REGION Network 33: Interface Signals 05 -Example: Model Flex-Pro-Line - IN/OUT- / Interface Signals 28
   // Aufruf des Schnittstellen Signal Bausteins Ba-Bereich 4 / Call the interface signals bool blocks of opmode 4
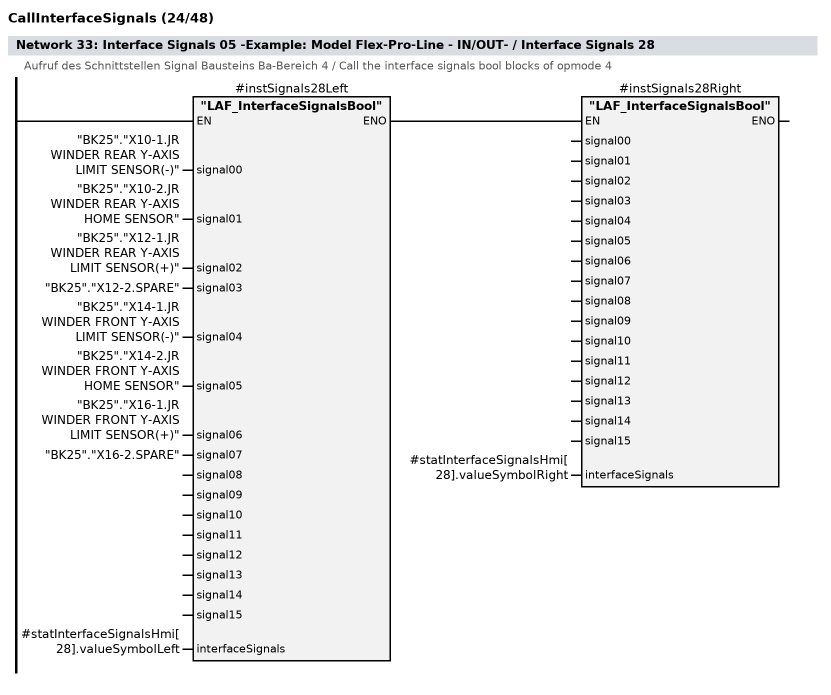
   RUNG wire#powerrail
      #instSignals28Left(signal00 := "BK25"."X10-1.JR WINDER REAR Y-AXIS LIMIT SENSOR(-)", signal01 := "BK25"."X10-2.JR WINDER REAR Y-AXIS HOME SENSOR", signal02 := "BK25"."X12-1.JR WINDER REAR Y-AXIS LIMIT SENSOR(+)", signal03 := "BK25"."X12-2.SPARE", signal04 := "BK25"."X14-1.JR WINDER FRONT Y-AXIS LIMIT SENSOR(-)", signal05 := "BK25"."X14-2.JR WINDER FRONT Y-AXIS HOME SENSOR", signal06 := "BK25"."X16-1.JR WINDER FRONT Y-AXIS LIMIT SENSOR(+)", signal07 := "BK25"."X16-2.SPARE", signal08 :=, signal09 :=, signal10 :=, signal11 :=, signal12 :=, signal13 :=, signal14 :=, signal15 :=, interfaceSignals := #statInterfaceSignalsHmi[28].valueSymbolLeft)
      #instSignals28Right(signal00 :=, signal01 :=, signal02 :=, signal03 :=, signal04 :=, signal05 :=, signal06 :=, signal07 :=, signal08 :=, signal09 :=, signal10 :=, signal11 :=, signal12 :=, signal13 :=, signal14 :=, signal15 :=, interfaceSignals := #statInterfaceSignalsHmi[28].valueSymbolRight)
   END_RUNG
   // the same network as SCL:
   #instSignals28Left(signal00 := "BK25"."X10-1.JR WINDER REAR Y-AXIS LIMIT SENSOR(-)",   // "LAF_InterfaceSignalsBool"
                      signal01 := "BK25"."X10-2.JR WINDER REAR Y-AXIS HOME SENSOR",
                      signal02 := "BK25"."X12-1.JR WINDER REAR Y-AXIS LIMIT SENSOR(+)",
                      signal03 := "BK25"."X12-2.SPARE",
                      signal04 := "BK25"."X14-1.JR WINDER FRONT Y-AXIS LIMIT SENSOR(-)",
                      signal05 := "BK25"."X14-2.JR WINDER FRONT Y-AXIS HOME SENSOR",
                      signal06 := "BK25"."X16-1.JR WINDER FRONT Y-AXIS LIMIT SENSOR(+)",
                      signal07 := "BK25"."X16-2.SPARE",
                      interfaceSignals := #statInterfaceSignalsHmi[28].valueSymbolLeft,
                      ENO => #_w1);
   IF #_w1 THEN
       #instSignals28Right(interfaceSignals := #statInterfaceSignalsHmi[28].valueSymbolRight);   // "LAF_InterfaceSignalsBool"
   END_IF;
END_REGION

REGION Network 34: Interface Signals 05 -Example: Model Flex-Pro-Line - IN/OUT- / Interface Signals 29
   // Aufruf des Schnittstellen Signal Bausteins Ba-Bereich 4 / Call the interface signals bool blocks of opmode 4
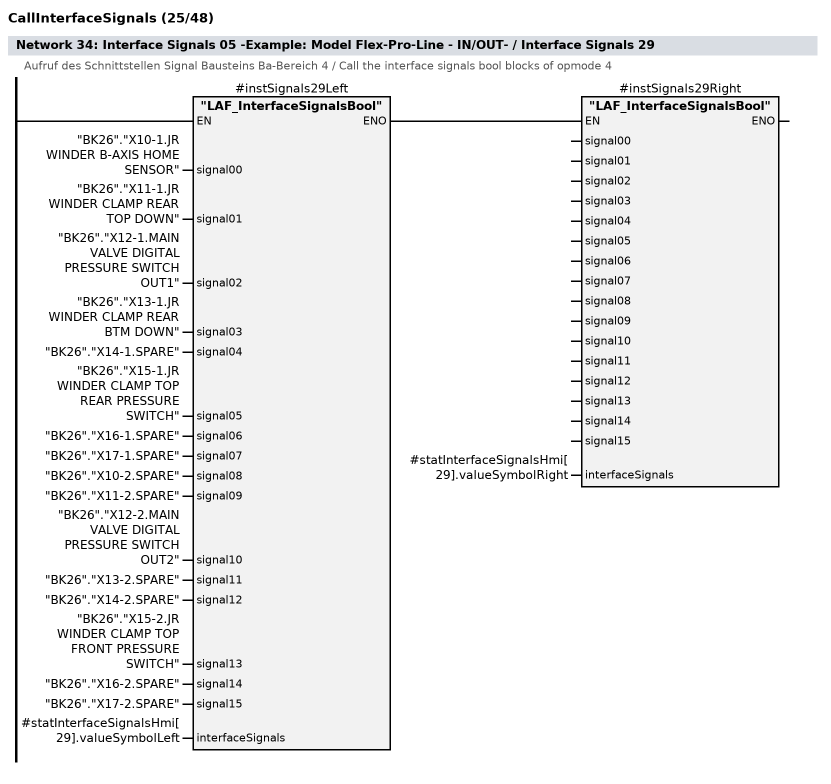
   RUNG wire#powerrail
      #instSignals29Left(signal00 := "BK26"."X10-1.JR WINDER B-AXIS HOME SENSOR", signal01 := "BK26"."X11-1.JR WINDER CLAMP REAR TOP DOWN", signal02 := "BK26"."X12-1.MAIN VALVE DIGITAL PRESSURE SWITCH OUT1", signal03 := "BK26"."X13-1.JR WINDER CLAMP REAR BTM DOWN", signal04 := "BK26"."X14-1.SPARE", signal05 := "BK26"."X15-1.JR WINDER CLAMP TOP REAR PRESSURE SWITCH", signal06 := "BK26"."X16-1.SPARE", signal07 := "BK26"."X17-1.SPARE", signal08 := "BK26"."X10-2.SPARE", signal09 := "BK26"."X11-2.SPARE", signal10 := "BK26"."X12-2.MAIN VALVE DIGITAL PRESSURE SWITCH OUT2", signal11 := "BK26"."X13-2.SPARE", signal12 := "BK26"."X14-2.SPARE", signal13 := "BK26"."X15-2.JR WINDER CLAMP TOP FRONT PRESSURE SWITCH", signal14 := "BK26"."X16-2.SPARE", signal15 := "BK26"."X17-2.SPARE", interfaceSignals := #statInterfaceSignalsHmi[29].valueSymbolLeft)
      #instSignals29Right(signal00 :=, signal01 :=, signal02 :=, signal03 :=, signal04 :=, signal05 :=, signal06 :=, signal07 :=, signal08 :=, signal09 :=, signal10 :=, signal11 :=, signal12 :=, signal13 :=, signal14 :=, signal15 :=, interfaceSignals := #statInterfaceSignalsHmi[29].valueSymbolRight)
   END_RUNG
   // the same network as SCL:
   #instSignals29Left(signal00 := "BK26"."X10-1.JR WINDER B-AXIS HOME SENSOR",   // "LAF_InterfaceSignalsBool"
                      signal01 := "BK26"."X11-1.JR WINDER CLAMP REAR TOP DOWN",
                      signal02 := "BK26"."X12-1.MAIN VALVE DIGITAL PRESSURE SWITCH OUT1",
                      signal03 := "BK26"."X13-1.JR WINDER CLAMP REAR BTM DOWN",
                      signal04 := "BK26"."X14-1.SPARE",
                      signal05 := "BK26"."X15-1.JR WINDER CLAMP TOP REAR PRESSURE SWITCH",
                      signal06 := "BK26"."X16-1.SPARE",
                      signal07 := "BK26"."X17-1.SPARE",
                      signal08 := "BK26"."X10-2.SPARE",
                      signal09 := "BK26"."X11-2.SPARE",
                      signal10 := "BK26"."X12-2.MAIN VALVE DIGITAL PRESSURE SWITCH OUT2",
                      signal11 := "BK26"."X13-2.SPARE",
                      signal12 := "BK26"."X14-2.SPARE",
                      signal13 := "BK26"."X15-2.JR WINDER CLAMP TOP FRONT PRESSURE SWITCH",
                      signal14 := "BK26"."X16-2.SPARE",
                      signal15 := "BK26"."X17-2.SPARE",
                      interfaceSignals := #statInterfaceSignalsHmi[29].valueSymbolLeft,
                      ENO => #_w1);
   IF #_w1 THEN
       #instSignals29Right(interfaceSignals := #statInterfaceSignalsHmi[29].valueSymbolRight);   // "LAF_InterfaceSignalsBool"
   END_IF;
END_REGION

REGION Network 35: Interface Signals 05 -Example: Model Flex-Pro-Line - IN/OUT- / Interface Signals 30
   // Aufruf des Schnittstellen Signal Bausteins Ba-Bereich 4 / Call the interface signals bool blocks of opmode 4
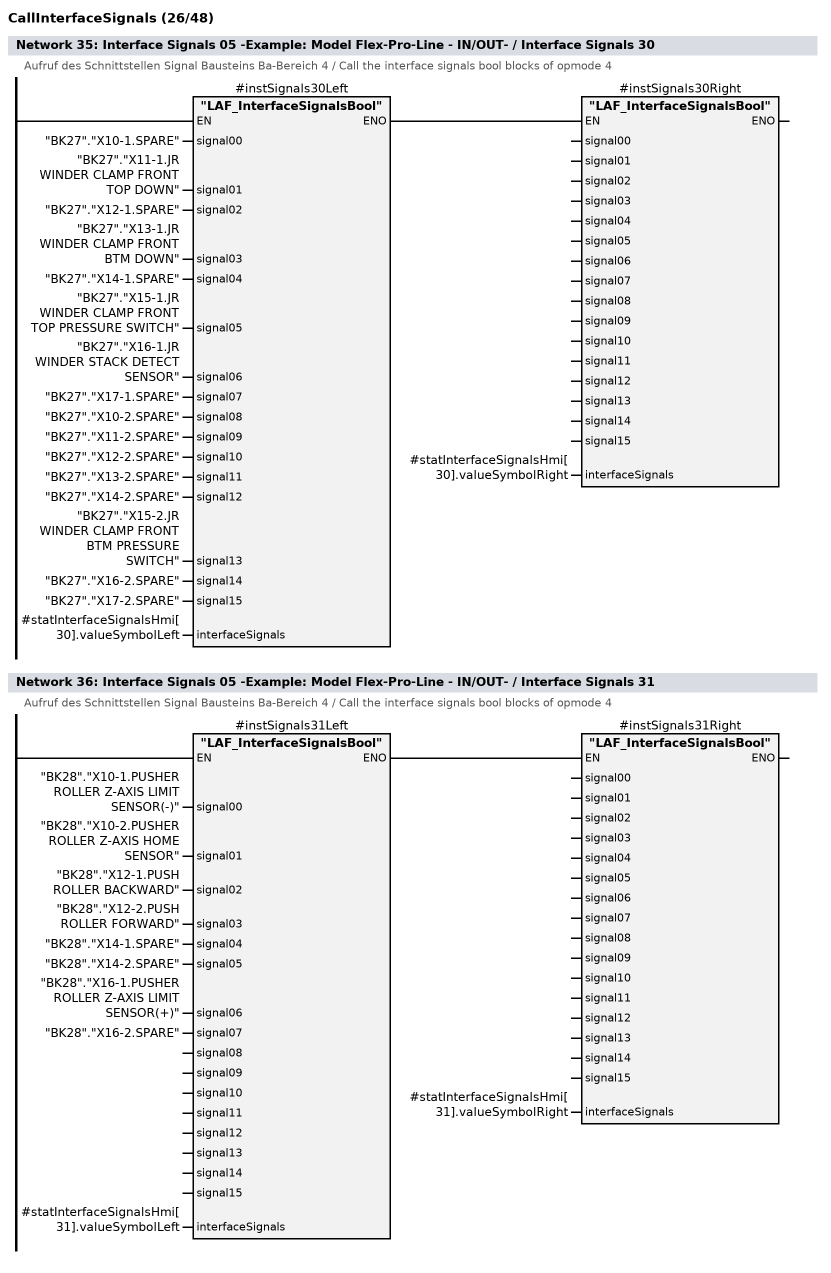
   RUNG wire#powerrail
      #instSignals30Left(signal00 := "BK27"."X10-1.SPARE", signal01 := "BK27"."X11-1.JR WINDER CLAMP FRONT TOP DOWN", signal02 := "BK27"."X12-1.SPARE", signal03 := "BK27"."X13-1.JR WINDER CLAMP FRONT BTM DOWN", signal04 := "BK27"."X14-1.SPARE", signal05 := "BK27"."X15-1.JR WINDER CLAMP FRONT TOP PRESSURE SWITCH", signal06 := "BK27"."X16-1.JR WINDER STACK DETECT SENSOR", signal07 := "BK27"."X17-1.SPARE", signal08 := "BK27"."X10-2.SPARE", signal09 := "BK27"."X11-2.SPARE", signal10 := "BK27"."X12-2.SPARE", signal11 := "BK27"."X13-2.SPARE", signal12 := "BK27"."X14-2.SPARE", signal13 := "BK27"."X15-2.JR WINDER CLAMP FRONT BTM PRESSURE SWITCH", signal14 := "BK27"."X16-2.SPARE", signal15 := "BK27"."X17-2.SPARE", interfaceSignals := #statInterfaceSignalsHmi[30].valueSymbolLeft)
      #instSignals30Right(signal00 :=, signal01 :=, signal02 :=, signal03 :=, signal04 :=, signal05 :=, signal06 :=, signal07 :=, signal08 :=, signal09 :=, signal10 :=, signal11 :=, signal12 :=, signal13 :=, signal14 :=, signal15 :=, interfaceSignals := #statInterfaceSignalsHmi[30].valueSymbolRight)
   END_RUNG
   // the same network as SCL:
   #instSignals30Left(signal00 := "BK27"."X10-1.SPARE",   // "LAF_InterfaceSignalsBool"
                      signal01 := "BK27"."X11-1.JR WINDER CLAMP FRONT TOP DOWN",
                      signal02 := "BK27"."X12-1.SPARE",
                      signal03 := "BK27"."X13-1.JR WINDER CLAMP FRONT BTM DOWN",
                      signal04 := "BK27"."X14-1.SPARE",
                      signal05 := "BK27"."X15-1.JR WINDER CLAMP FRONT TOP PRESSURE SWITCH",
                      signal06 := "BK27"."X16-1.JR WINDER STACK DETECT SENSOR",
                      signal07 := "BK27"."X17-1.SPARE",
                      signal08 := "BK27"."X10-2.SPARE",
                      signal09 := "BK27"."X11-2.SPARE",
                      signal10 := "BK27"."X12-2.SPARE",
                      signal11 := "BK27"."X13-2.SPARE",
                      signal12 := "BK27"."X14-2.SPARE",
                      signal13 := "BK27"."X15-2.JR WINDER CLAMP FRONT BTM PRESSURE SWITCH",
                      signal14 := "BK27"."X16-2.SPARE",
                      signal15 := "BK27"."X17-2.SPARE",
                      interfaceSignals := #statInterfaceSignalsHmi[30].valueSymbolLeft,
                      ENO => #_w1);
   IF #_w1 THEN
       #instSignals30Right(interfaceSignals := #statInterfaceSignalsHmi[30].valueSymbolRight);   // "LAF_InterfaceSignalsBool"
   END_IF;
END_REGION

REGION Network 36: Interface Signals 05 -Example: Model Flex-Pro-Line - IN/OUT- / Interface Signals 31
   // Aufruf des Schnittstellen Signal Bausteins Ba-Bereich 4 / Call the interface signals bool blocks of opmode 4
   RUNG wire#powerrail
      #instSignals31Left(signal00 := "BK28"."X10-1.PUSHER ROLLER Z-AXIS LIMIT SENSOR(-)", signal01 := "BK28"."X10-2.PUSHER ROLLER Z-AXIS HOME SENSOR", signal02 := "BK28"."X12-1.PUSH ROLLER BACKWARD", signal03 := "BK28"."X12-2.PUSH ROLLER FORWARD", signal04 := "BK28"."X14-1.SPARE", signal05 := "BK28"."X14-2.SPARE", signal06 := "BK28"."X16-1.PUSHER ROLLER Z-AXIS LIMIT SENSOR(+)", signal07 := "BK28"."X16-2.SPARE", signal08 :=, signal09 :=, signal10 :=, signal11 :=, signal12 :=, signal13 :=, signal14 :=, signal15 :=, interfaceSignals := #statInterfaceSignalsHmi[31].valueSymbolLeft)
      #instSignals31Right(signal00 :=, signal01 :=, signal02 :=, signal03 :=, signal04 :=, signal05 :=, signal06 :=, signal07 :=, signal08 :=, signal09 :=, signal10 :=, signal11 :=, signal12 :=, signal13 :=, signal14 :=, signal15 :=, interfaceSignals := #statInterfaceSignalsHmi[31].valueSymbolRight)
   END_RUNG
   // the same network as SCL:
   #instSignals31Left(signal00 := "BK28"."X10-1.PUSHER ROLLER Z-AXIS LIMIT SENSOR(-)",   // "LAF_InterfaceSignalsBool"
                      signal01 := "BK28"."X10-2.PUSHER ROLLER Z-AXIS HOME SENSOR",
                      signal02 := "BK28"."X12-1.PUSH ROLLER BACKWARD",
                      signal03 := "BK28"."X12-2.PUSH ROLLER FORWARD",
                      signal04 := "BK28"."X14-1.SPARE",
                      signal05 := "BK28"."X14-2.SPARE",
                      signal06 := "BK28"."X16-1.PUSHER ROLLER Z-AXIS LIMIT SENSOR(+)",
                      signal07 := "BK28"."X16-2.SPARE",
                      interfaceSignals := #statInterfaceSignalsHmi[31].valueSymbolLeft,
                      ENO => #_w1);
   IF #_w1 THEN
       #instSignals31Right(interfaceSignals := #statInterfaceSignalsHmi[31].valueSymbolRight);   // "LAF_InterfaceSignalsBool"
   END_IF;
END_REGION

REGION Network 37: Interface Signals 05 -Example: Model Flex-Pro-Line - IN/OUT- / Interface Signals 32
   // Aufruf des Schnittstellen Signal Bausteins Ba-Bereich 4 / Call the interface signals bool blocks of opmode 4
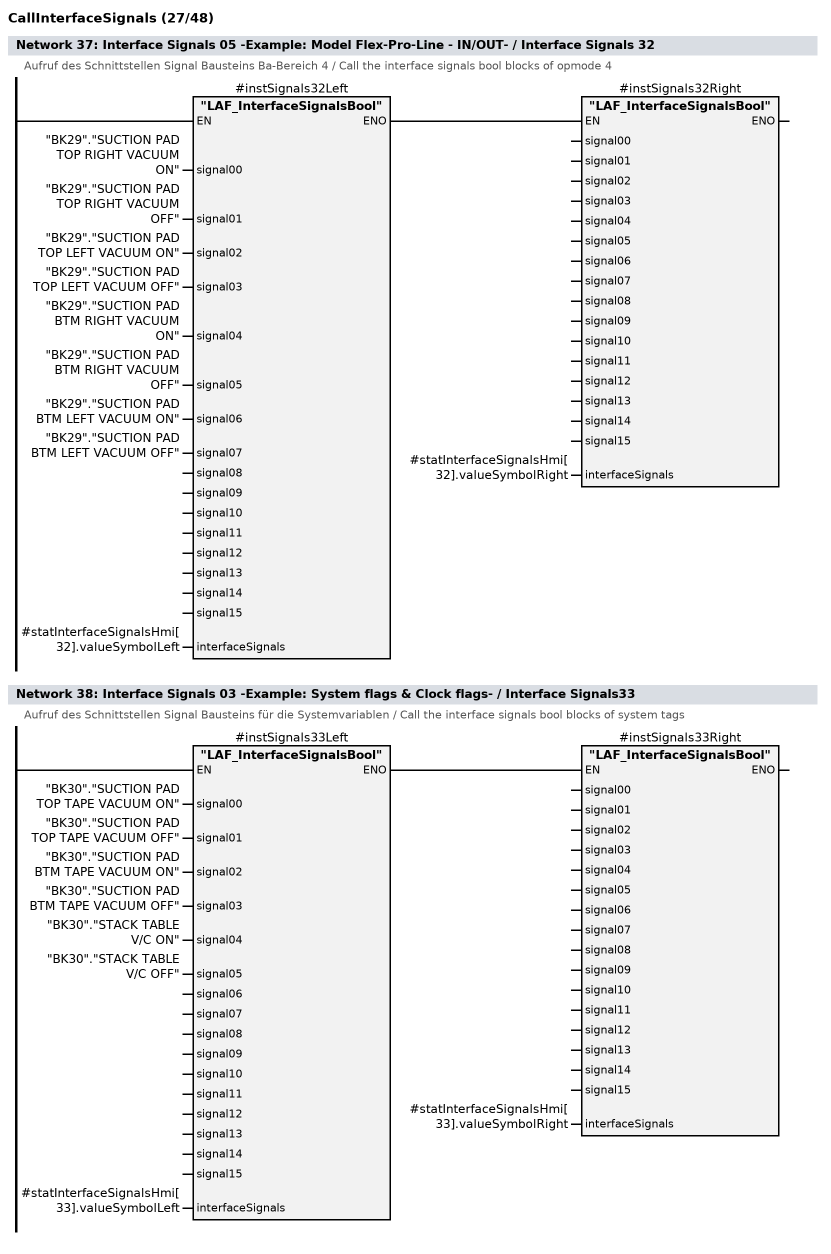
   RUNG wire#powerrail
      #instSignals32Left(signal00 := "BK29"."SUCTION PAD TOP RIGHT VACUUM ON", signal01 := "BK29"."SUCTION PAD TOP RIGHT VACUUM OFF", signal02 := "BK29"."SUCTION PAD TOP LEFT VACUUM ON", signal03 := "BK29"."SUCTION PAD TOP LEFT VACUUM OFF", signal04 := "BK29"."SUCTION PAD BTM RIGHT VACUUM ON", signal05 := "BK29"."SUCTION PAD BTM RIGHT VACUUM OFF", signal06 := "BK29"."SUCTION PAD BTM LEFT VACUUM ON", signal07 := "BK29"."SUCTION PAD BTM LEFT VACUUM OFF", signal08 :=, signal09 :=, signal10 :=, signal11 :=, signal12 :=, signal13 :=, signal14 :=, signal15 :=, interfaceSignals := #statInterfaceSignalsHmi[32].valueSymbolLeft)
      #instSignals32Right(signal00 :=, signal01 :=, signal02 :=, signal03 :=, signal04 :=, signal05 :=, signal06 :=, signal07 :=, signal08 :=, signal09 :=, signal10 :=, signal11 :=, signal12 :=, signal13 :=, signal14 :=, signal15 :=, interfaceSignals := #statInterfaceSignalsHmi[32].valueSymbolRight)
   END_RUNG
   // the same network as SCL:
   #instSignals32Left(signal00 := "BK29"."SUCTION PAD TOP RIGHT VACUUM ON",   // "LAF_InterfaceSignalsBool"
                      signal01 := "BK29"."SUCTION PAD TOP RIGHT VACUUM OFF",
                      signal02 := "BK29"."SUCTION PAD TOP LEFT VACUUM ON",
                      signal03 := "BK29"."SUCTION PAD TOP LEFT VACUUM OFF",
                      signal04 := "BK29"."SUCTION PAD BTM RIGHT VACUUM ON",
                      signal05 := "BK29"."SUCTION PAD BTM RIGHT VACUUM OFF",
                      signal06 := "BK29"."SUCTION PAD BTM LEFT VACUUM ON",
                      signal07 := "BK29"."SUCTION PAD BTM LEFT VACUUM OFF",
                      interfaceSignals := #statInterfaceSignalsHmi[32].valueSymbolLeft,
                      ENO => #_w1);
   IF #_w1 THEN
       #instSignals32Right(interfaceSignals := #statInterfaceSignalsHmi[32].valueSymbolRight);   // "LAF_InterfaceSignalsBool"
   END_IF;
END_REGION

REGION Network 38: Interface Signals 03 -Example: System flags & Clock flags- / Interface Signals33
   // Aufruf des Schnittstellen Signal Bausteins für die Systemvariablen / Call the interface signals bool blocks of system tags
   RUNG wire#powerrail
      #instSignals33Left(signal00 := "BK30"."SUCTION PAD TOP TAPE VACUUM ON", signal01 := "BK30"."SUCTION PAD TOP TAPE VACUUM OFF", signal02 := "BK30"."SUCTION PAD BTM TAPE VACUUM ON", signal03 := "BK30"."SUCTION PAD BTM TAPE VACUUM OFF", signal04 := "BK30"."STACK TABLE V/C ON", signal05 := "BK30"."STACK TABLE V/C OFF", signal06 :=, signal07 :=, signal08 :=, signal09 :=, signal10 :=, signal11 :=, signal12 :=, signal13 :=, signal14 :=, signal15 :=, interfaceSignals := #statInterfaceSignalsHmi[33].valueSymbolLeft)
      #instSignals33Right(signal00 :=, signal01 :=, signal02 :=, signal03 :=, signal04 :=, signal05 :=, signal06 :=, signal07 :=, signal08 :=, signal09 :=, signal10 :=, signal11 :=, signal12 :=, signal13 :=, signal14 :=, signal15 :=, interfaceSignals := #statInterfaceSignalsHmi[33].valueSymbolRight)
   END_RUNG
   // the same network as SCL:
   #instSignals33Left(signal00 := "BK30"."SUCTION PAD TOP TAPE VACUUM ON",   // "LAF_InterfaceSignalsBool"
                      signal01 := "BK30"."SUCTION PAD TOP TAPE VACUUM OFF",
                      signal02 := "BK30"."SUCTION PAD BTM TAPE VACUUM ON",
                      signal03 := "BK30"."SUCTION PAD BTM TAPE VACUUM OFF",
                      signal04 := "BK30"."STACK TABLE V/C ON",
                      signal05 := "BK30"."STACK TABLE V/C OFF",
                      interfaceSignals := #statInterfaceSignalsHmi[33].valueSymbolLeft,
                      ENO => #_w1);
   IF #_w1 THEN
       #instSignals33Right(interfaceSignals := #statInterfaceSignalsHmi[33].valueSymbolRight);   // "LAF_InterfaceSignalsBool"
   END_IF;
END_REGION

REGION Network 39: Interface Signals 04 -Example: Model Flex-Pro-Line - IN/OUT- / Interface Signals 34
   // Aufruf des Schnittstellen Signal Bausteins Ba-Bereich 4 / Call the interface signals bool blocks of opmode 4
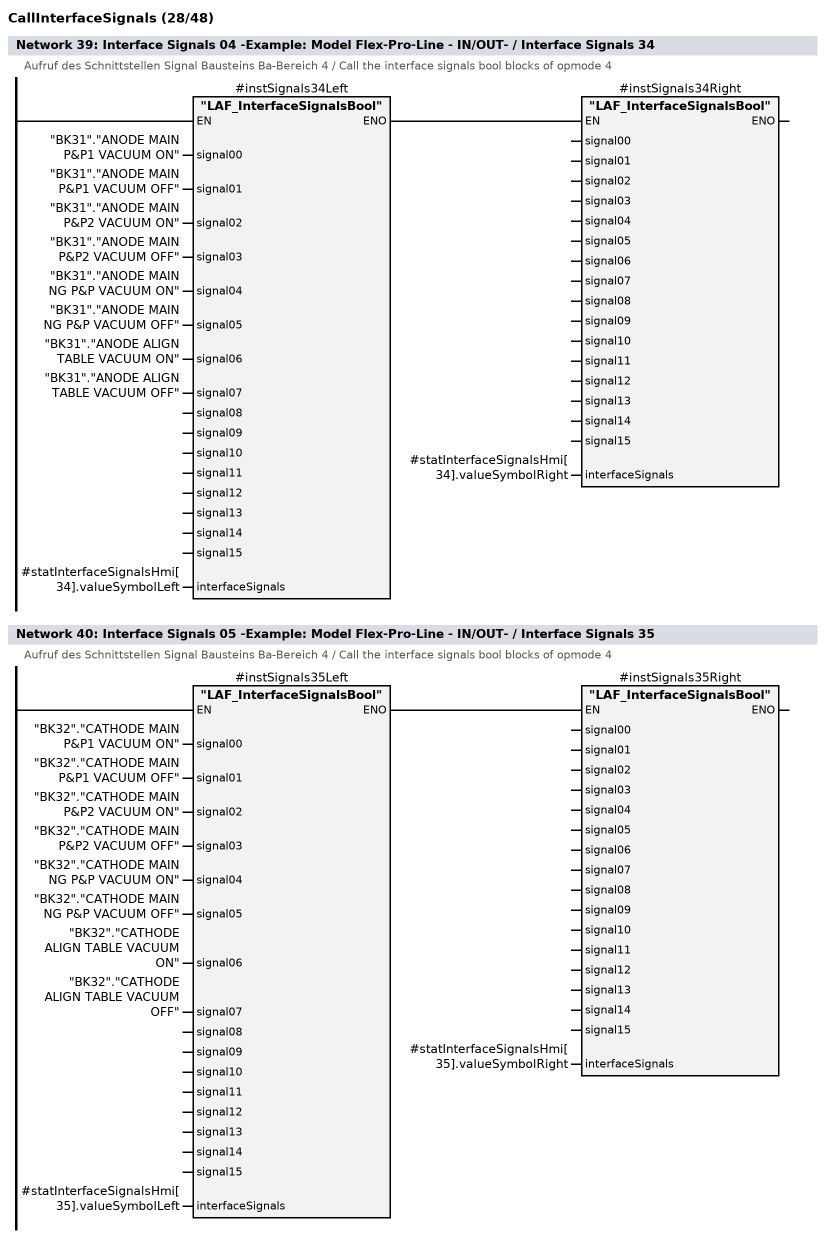
   RUNG wire#powerrail
      #instSignals34Left(signal00 := "BK31"."ANODE MAIN P&P1 VACUUM ON", signal01 := "BK31"."ANODE MAIN P&P1 VACUUM OFF", signal02 := "BK31"."ANODE MAIN P&P2 VACUUM ON", signal03 := "BK31"."ANODE MAIN P&P2 VACUUM OFF", signal04 := "BK31"."ANODE MAIN NG P&P VACUUM ON", signal05 := "BK31"."ANODE MAIN NG P&P VACUUM OFF", signal06 := "BK31"."ANODE ALIGN TABLE VACUUM ON", signal07 := "BK31"."ANODE ALIGN TABLE VACUUM OFF", signal08 :=, signal09 :=, signal10 :=, signal11 :=, signal12 :=, signal13 :=, signal14 :=, signal15 :=, interfaceSignals := #statInterfaceSignalsHmi[34].valueSymbolLeft)
      #instSignals34Right(signal00 :=, signal01 :=, signal02 :=, signal03 :=, signal04 :=, signal05 :=, signal06 :=, signal07 :=, signal08 :=, signal09 :=, signal10 :=, signal11 :=, signal12 :=, signal13 :=, signal14 :=, signal15 :=, interfaceSignals := #statInterfaceSignalsHmi[34].valueSymbolRight)
   END_RUNG
   // the same network as SCL:
   #instSignals34Left(signal00 := "BK31"."ANODE MAIN P&P1 VACUUM ON",   // "LAF_InterfaceSignalsBool"
                      signal01 := "BK31"."ANODE MAIN P&P1 VACUUM OFF",
                      signal02 := "BK31"."ANODE MAIN P&P2 VACUUM ON",
                      signal03 := "BK31"."ANODE MAIN P&P2 VACUUM OFF",
                      signal04 := "BK31"."ANODE MAIN NG P&P VACUUM ON",
                      signal05 := "BK31"."ANODE MAIN NG P&P VACUUM OFF",
                      signal06 := "BK31"."ANODE ALIGN TABLE VACUUM ON",
                      signal07 := "BK31"."ANODE ALIGN TABLE VACUUM OFF",
                      interfaceSignals := #statInterfaceSignalsHmi[34].valueSymbolLeft,
                      ENO => #_w1);
   IF #_w1 THEN
       #instSignals34Right(interfaceSignals := #statInterfaceSignalsHmi[34].valueSymbolRight);   // "LAF_InterfaceSignalsBool"
   END_IF;
END_REGION

REGION Network 40: Interface Signals 05 -Example: Model Flex-Pro-Line - IN/OUT- / Interface Signals 35
   // Aufruf des Schnittstellen Signal Bausteins Ba-Bereich 4 / Call the interface signals bool blocks of opmode 4
   RUNG wire#powerrail
      #instSignals35Left(signal00 := "BK32"."CATHODE MAIN P&P1 VACUUM ON", signal01 := "BK32"."CATHODE MAIN P&P1 VACUUM OFF", signal02 := "BK32"."CATHODE MAIN P&P2 VACUUM ON", signal03 := "BK32"."CATHODE MAIN P&P2 VACUUM OFF", signal04 := "BK32"."CATHODE MAIN NG P&P VACUUM ON", signal05 := "BK32"."CATHODE MAIN NG P&P VACUUM OFF", signal06 := "BK32"."CATHODE ALIGN TABLE VACUUM ON", signal07 := "BK32"."CATHODE ALIGN TABLE VACUUM OFF", signal08 :=, signal09 :=, signal10 :=, signal11 :=, signal12 :=, signal13 :=, signal14 :=, signal15 :=, interfaceSignals := #statInterfaceSignalsHmi[35].valueSymbolLeft)
      #instSignals35Right(signal00 :=, signal01 :=, signal02 :=, signal03 :=, signal04 :=, signal05 :=, signal06 :=, signal07 :=, signal08 :=, signal09 :=, signal10 :=, signal11 :=, signal12 :=, signal13 :=, signal14 :=, signal15 :=, interfaceSignals := #statInterfaceSignalsHmi[35].valueSymbolRight)
   END_RUNG
   // the same network as SCL:
   #instSignals35Left(signal00 := "BK32"."CATHODE MAIN P&P1 VACUUM ON",   // "LAF_InterfaceSignalsBool"
                      signal01 := "BK32"."CATHODE MAIN P&P1 VACUUM OFF",
                      signal02 := "BK32"."CATHODE MAIN P&P2 VACUUM ON",
                      signal03 := "BK32"."CATHODE MAIN P&P2 VACUUM OFF",
                      signal04 := "BK32"."CATHODE MAIN NG P&P VACUUM ON",
                      signal05 := "BK32"."CATHODE MAIN NG P&P VACUUM OFF",
                      signal06 := "BK32"."CATHODE ALIGN TABLE VACUUM ON",
                      signal07 := "BK32"."CATHODE ALIGN TABLE VACUUM OFF",
                      interfaceSignals := #statInterfaceSignalsHmi[35].valueSymbolLeft,
                      ENO => #_w1);
   IF #_w1 THEN
       #instSignals35Right(interfaceSignals := #statInterfaceSignalsHmi[35].valueSymbolRight);   // "LAF_InterfaceSignalsBool"
   END_IF;
END_REGION

REGION Network 41: Interface Signals 05 -Example: Model Flex-Pro-Line - IN/OUT- / Interface Signals 36
   // Aufruf des Schnittstellen Signal Bausteins Ba-Bereich 4 / Call the interface signals bool blocks of opmode 4
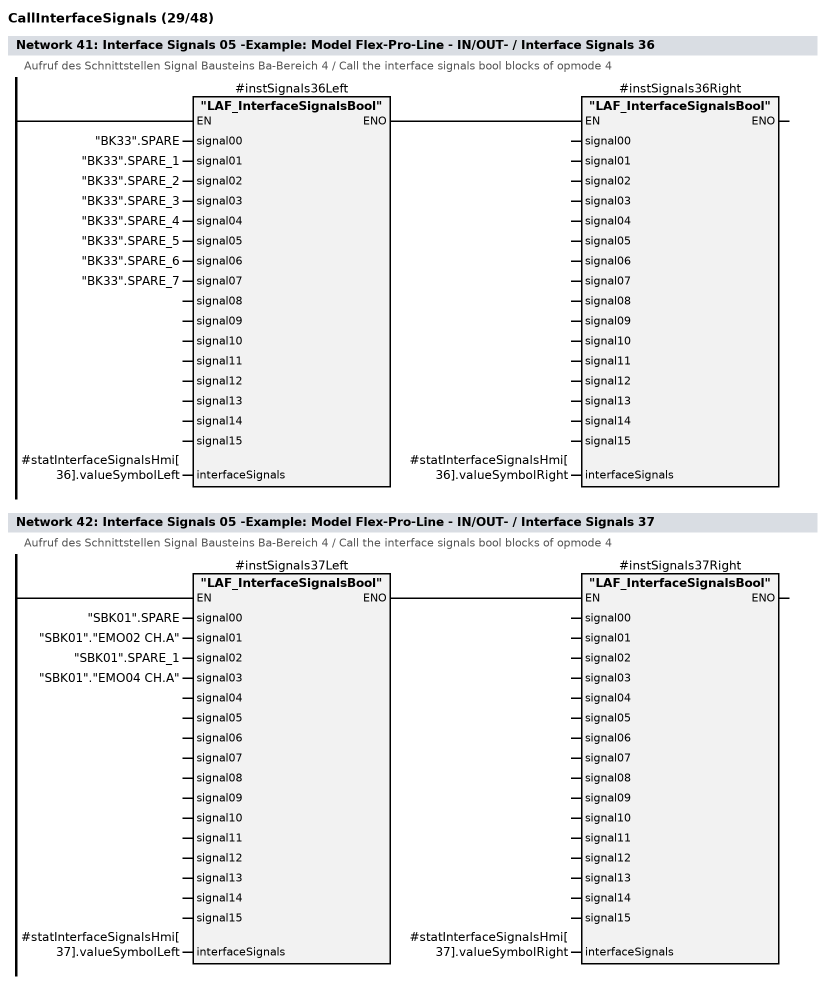
   RUNG wire#powerrail
      #instSignals36Left(signal00 := "BK33".SPARE, signal01 := "BK33".SPARE_1, signal02 := "BK33".SPARE_2, signal03 := "BK33".SPARE_3, signal04 := "BK33".SPARE_4, signal05 := "BK33".SPARE_5, signal06 := "BK33".SPARE_6, signal07 := "BK33".SPARE_7, signal08 :=, signal09 :=, signal10 :=, signal11 :=, signal12 :=, signal13 :=, signal14 :=, signal15 :=, interfaceSignals := #statInterfaceSignalsHmi[36].valueSymbolLeft)
      #instSignals36Right(signal00 :=, signal01 :=, signal02 :=, signal03 :=, signal04 :=, signal05 :=, signal06 :=, signal07 :=, signal08 :=, signal09 :=, signal10 :=, signal11 :=, signal12 :=, signal13 :=, signal14 :=, signal15 :=, interfaceSignals := #statInterfaceSignalsHmi[36].valueSymbolRight)
   END_RUNG
   // the same network as SCL:
   #instSignals36Left(signal00 := "BK33".SPARE,   // "LAF_InterfaceSignalsBool"
                      signal01 := "BK33".SPARE_1,
                      signal02 := "BK33".SPARE_2,
                      signal03 := "BK33".SPARE_3,
                      signal04 := "BK33".SPARE_4,
                      signal05 := "BK33".SPARE_5,
                      signal06 := "BK33".SPARE_6,
                      signal07 := "BK33".SPARE_7,
                      interfaceSignals := #statInterfaceSignalsHmi[36].valueSymbolLeft,
                      ENO => #_w1);
   IF #_w1 THEN
       #instSignals36Right(interfaceSignals := #statInterfaceSignalsHmi[36].valueSymbolRight);   // "LAF_InterfaceSignalsBool"
   END_IF;
END_REGION

REGION Network 42: Interface Signals 05 -Example: Model Flex-Pro-Line - IN/OUT- / Interface Signals 37
   // Aufruf des Schnittstellen Signal Bausteins Ba-Bereich 4 / Call the interface signals bool blocks of opmode 4
   RUNG wire#powerrail
      #instSignals37Left(signal00 := "SBK01".SPARE, signal01 := "SBK01"."EMO02 CH.A", signal02 := "SBK01".SPARE_1, signal03 := "SBK01"."EMO04 CH.A", signal04 :=, signal05 :=, signal06 :=, signal07 :=, signal08 :=, signal09 :=, signal10 :=, signal11 :=, signal12 :=, signal13 :=, signal14 :=, signal15 :=, interfaceSignals := #statInterfaceSignalsHmi[37].valueSymbolLeft)
      #instSignals37Right(signal00 :=, signal01 :=, signal02 :=, signal03 :=, signal04 :=, signal05 :=, signal06 :=, signal07 :=, signal08 :=, signal09 :=, signal10 :=, signal11 :=, signal12 :=, signal13 :=, signal14 :=, signal15 :=, interfaceSignals := #statInterfaceSignalsHmi[37].valueSymbolRight)
   END_RUNG
   // the same network as SCL:
   #instSignals37Left(signal00 := "SBK01".SPARE,   // "LAF_InterfaceSignalsBool"
                      signal01 := "SBK01"."EMO02 CH.A",
                      signal02 := "SBK01".SPARE_1,
                      signal03 := "SBK01"."EMO04 CH.A",
                      interfaceSignals := #statInterfaceSignalsHmi[37].valueSymbolLeft,
                      ENO => #_w1);
   IF #_w1 THEN
       #instSignals37Right(interfaceSignals := #statInterfaceSignalsHmi[37].valueSymbolRight);   // "LAF_InterfaceSignalsBool"
   END_IF;
END_REGION

REGION Network 43: Interface Signals 05 -Example: Model Flex-Pro-Line - IN/OUT- / Interface Signals 38
   // Aufruf des Schnittstellen Signal Bausteins Ba-Bereich 4 / Call the interface signals bool blocks of opmode 4
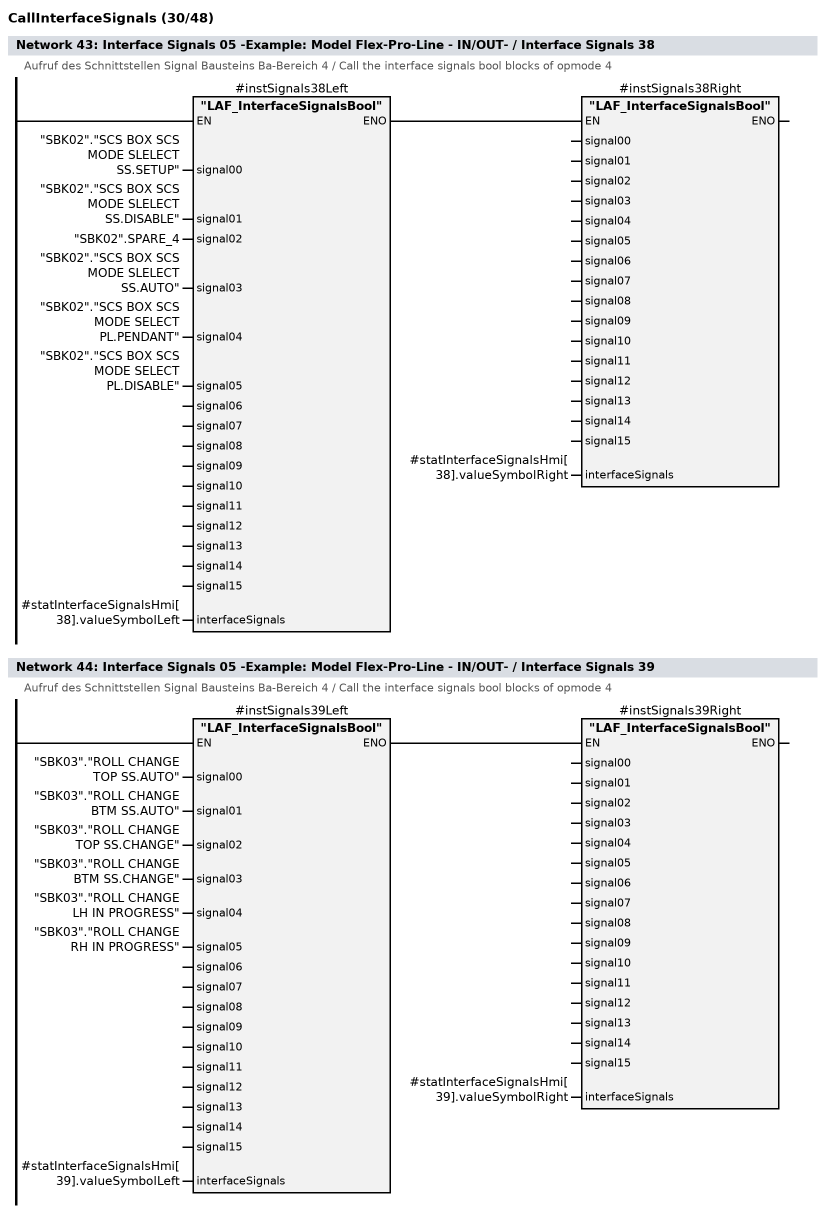
   RUNG wire#powerrail
      #instSignals38Left(signal00 := "SBK02"."SCS BOX SCS MODE SLELECT SS.SETUP", signal01 := "SBK02"."SCS BOX SCS MODE SLELECT SS.DISABLE", signal02 := "SBK02".SPARE_4, signal03 := "SBK02"."SCS BOX SCS MODE SLELECT SS.AUTO", signal04 := "SBK02"."SCS BOX SCS MODE SELECT PL.PENDANT", signal05 := "SBK02"."SCS BOX SCS MODE SELECT PL.DISABLE", signal06 :=, signal07 :=, signal08 :=, signal09 :=, signal10 :=, signal11 :=, signal12 :=, signal13 :=, signal14 :=, signal15 :=, interfaceSignals := #statInterfaceSignalsHmi[38].valueSymbolLeft)
      #instSignals38Right(signal00 :=, signal01 :=, signal02 :=, signal03 :=, signal04 :=, signal05 :=, signal06 :=, signal07 :=, signal08 :=, signal09 :=, signal10 :=, signal11 :=, signal12 :=, signal13 :=, signal14 :=, signal15 :=, interfaceSignals := #statInterfaceSignalsHmi[38].valueSymbolRight)
   END_RUNG
   // the same network as SCL:
   #instSignals38Left(signal00 := "SBK02"."SCS BOX SCS MODE SLELECT SS.SETUP",   // "LAF_InterfaceSignalsBool"
                      signal01 := "SBK02"."SCS BOX SCS MODE SLELECT SS.DISABLE",
                      signal02 := "SBK02".SPARE_4,
                      signal03 := "SBK02"."SCS BOX SCS MODE SLELECT SS.AUTO",
                      signal04 := "SBK02"."SCS BOX SCS MODE SELECT PL.PENDANT",
                      signal05 := "SBK02"."SCS BOX SCS MODE SELECT PL.DISABLE",
                      interfaceSignals := #statInterfaceSignalsHmi[38].valueSymbolLeft,
                      ENO => #_w1);
   IF #_w1 THEN
       #instSignals38Right(interfaceSignals := #statInterfaceSignalsHmi[38].valueSymbolRight);   // "LAF_InterfaceSignalsBool"
   END_IF;
END_REGION

REGION Network 44: Interface Signals 05 -Example: Model Flex-Pro-Line - IN/OUT- / Interface Signals 39
   // Aufruf des Schnittstellen Signal Bausteins Ba-Bereich 4 / Call the interface signals bool blocks of opmode 4
   RUNG wire#powerrail
      #instSignals39Left(signal00 := "SBK03"."ROLL CHANGE TOP SS.AUTO", signal01 := "SBK03"."ROLL CHANGE BTM SS.AUTO", signal02 := "SBK03"."ROLL CHANGE TOP SS.CHANGE", signal03 := "SBK03"."ROLL CHANGE BTM SS.CHANGE", signal04 := "SBK03"."ROLL CHANGE LH IN PROGRESS", signal05 := "SBK03"."ROLL CHANGE RH IN PROGRESS", signal06 :=, signal07 :=, signal08 :=, signal09 :=, signal10 :=, signal11 :=, signal12 :=, signal13 :=, signal14 :=, signal15 :=, interfaceSignals := #statInterfaceSignalsHmi[39].valueSymbolLeft)
      #instSignals39Right(signal00 :=, signal01 :=, signal02 :=, signal03 :=, signal04 :=, signal05 :=, signal06 :=, signal07 :=, signal08 :=, signal09 :=, signal10 :=, signal11 :=, signal12 :=, signal13 :=, signal14 :=, signal15 :=, interfaceSignals := #statInterfaceSignalsHmi[39].valueSymbolRight)
   END_RUNG
   // the same network as SCL:
   #instSignals39Left(signal00 := "SBK03"."ROLL CHANGE TOP SS.AUTO",   // "LAF_InterfaceSignalsBool"
                      signal01 := "SBK03"."ROLL CHANGE BTM SS.AUTO",
                      signal02 := "SBK03"."ROLL CHANGE TOP SS.CHANGE",
                      signal03 := "SBK03"."ROLL CHANGE BTM SS.CHANGE",
                      signal04 := "SBK03"."ROLL CHANGE LH IN PROGRESS",
                      signal05 := "SBK03"."ROLL CHANGE RH IN PROGRESS",
                      interfaceSignals := #statInterfaceSignalsHmi[39].valueSymbolLeft,
                      ENO => #_w1);
   IF #_w1 THEN
       #instSignals39Right(interfaceSignals := #statInterfaceSignalsHmi[39].valueSymbolRight);   // "LAF_InterfaceSignalsBool"
   END_IF;
END_REGION

REGION Network 45: Interface Signals 05 -Example: Model Flex-Pro-Line - IN/OUT- / Interface Signals 40
   // Aufruf des Schnittstellen Signal Bausteins Ba-Bereich 4 / Call the interface signals bool blocks of opmode 4
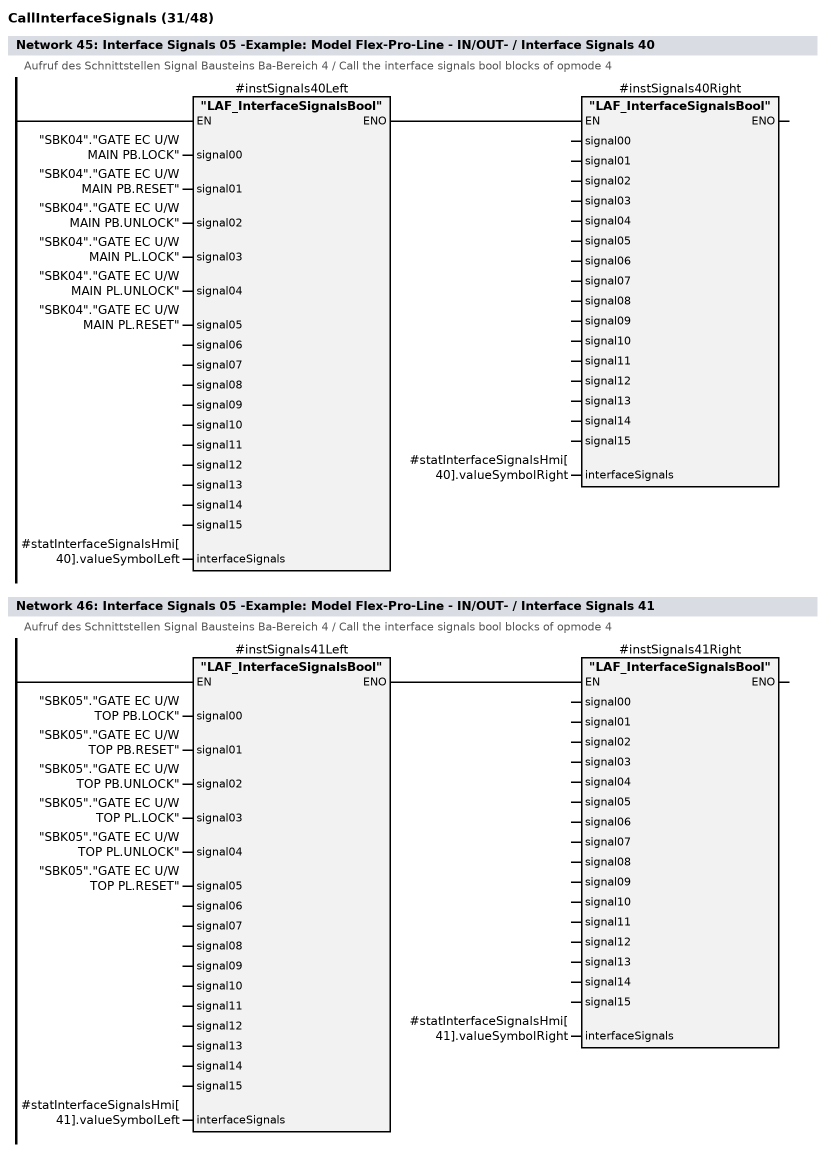
   RUNG wire#powerrail
      #instSignals40Left(signal00 := "SBK04"."GATE EC U/W MAIN PB.LOCK", signal01 := "SBK04"."GATE EC U/W MAIN PB.RESET", signal02 := "SBK04"."GATE EC U/W MAIN PB.UNLOCK", signal03 := "SBK04"."GATE EC U/W MAIN PL.LOCK", signal04 := "SBK04"."GATE EC U/W MAIN PL.UNLOCK", signal05 := "SBK04"."GATE EC U/W MAIN PL.RESET", signal06 :=, signal07 :=, signal08 :=, signal09 :=, signal10 :=, signal11 :=, signal12 :=, signal13 :=, signal14 :=, signal15 :=, interfaceSignals := #statInterfaceSignalsHmi[40].valueSymbolLeft)
      #instSignals40Right(signal00 :=, signal01 :=, signal02 :=, signal03 :=, signal04 :=, signal05 :=, signal06 :=, signal07 :=, signal08 :=, signal09 :=, signal10 :=, signal11 :=, signal12 :=, signal13 :=, signal14 :=, signal15 :=, interfaceSignals := #statInterfaceSignalsHmi[40].valueSymbolRight)
   END_RUNG
   // the same network as SCL:
   #instSignals40Left(signal00 := "SBK04"."GATE EC U/W MAIN PB.LOCK",   // "LAF_InterfaceSignalsBool"
                      signal01 := "SBK04"."GATE EC U/W MAIN PB.RESET",
                      signal02 := "SBK04"."GATE EC U/W MAIN PB.UNLOCK",
                      signal03 := "SBK04"."GATE EC U/W MAIN PL.LOCK",
                      signal04 := "SBK04"."GATE EC U/W MAIN PL.UNLOCK",
                      signal05 := "SBK04"."GATE EC U/W MAIN PL.RESET",
                      interfaceSignals := #statInterfaceSignalsHmi[40].valueSymbolLeft,
                      ENO => #_w1);
   IF #_w1 THEN
       #instSignals40Right(interfaceSignals := #statInterfaceSignalsHmi[40].valueSymbolRight);   // "LAF_InterfaceSignalsBool"
   END_IF;
END_REGION

REGION Network 46: Interface Signals 05 -Example: Model Flex-Pro-Line - IN/OUT- / Interface Signals 41
   // Aufruf des Schnittstellen Signal Bausteins Ba-Bereich 4 / Call the interface signals bool blocks of opmode 4
   RUNG wire#powerrail
      #instSignals41Left(signal00 := "SBK05"."GATE EC U/W TOP PB.LOCK", signal01 := "SBK05"."GATE EC U/W TOP PB.RESET", signal02 := "SBK05"."GATE EC U/W TOP PB.UNLOCK", signal03 := "SBK05"."GATE EC U/W TOP PL.LOCK", signal04 := "SBK05"."GATE EC U/W TOP PL.UNLOCK", signal05 := "SBK05"."GATE EC U/W TOP PL.RESET", signal06 :=, signal07 :=, signal08 :=, signal09 :=, signal10 :=, signal11 :=, signal12 :=, signal13 :=, signal14 :=, signal15 :=, interfaceSignals := #statInterfaceSignalsHmi[41].valueSymbolLeft)
      #instSignals41Right(signal00 :=, signal01 :=, signal02 :=, signal03 :=, signal04 :=, signal05 :=, signal06 :=, signal07 :=, signal08 :=, signal09 :=, signal10 :=, signal11 :=, signal12 :=, signal13 :=, signal14 :=, signal15 :=, interfaceSignals := #statInterfaceSignalsHmi[41].valueSymbolRight)
   END_RUNG
   // the same network as SCL:
   #instSignals41Left(signal00 := "SBK05"."GATE EC U/W TOP PB.LOCK",   // "LAF_InterfaceSignalsBool"
                      signal01 := "SBK05"."GATE EC U/W TOP PB.RESET",
                      signal02 := "SBK05"."GATE EC U/W TOP PB.UNLOCK",
                      signal03 := "SBK05"."GATE EC U/W TOP PL.LOCK",
                      signal04 := "SBK05"."GATE EC U/W TOP PL.UNLOCK",
                      signal05 := "SBK05"."GATE EC U/W TOP PL.RESET",
                      interfaceSignals := #statInterfaceSignalsHmi[41].valueSymbolLeft,
                      ENO => #_w1);
   IF #_w1 THEN
       #instSignals41Right(interfaceSignals := #statInterfaceSignalsHmi[41].valueSymbolRight);   // "LAF_InterfaceSignalsBool"
   END_IF;
END_REGION

REGION Network 47: Interface Signals 05 -Example: Model Flex-Pro-Line - IN/OUT- / Interface Signals 42
   // Aufruf des Schnittstellen Signal Bausteins Ba-Bereich 4 / Call the interface signals bool blocks of opmode 4
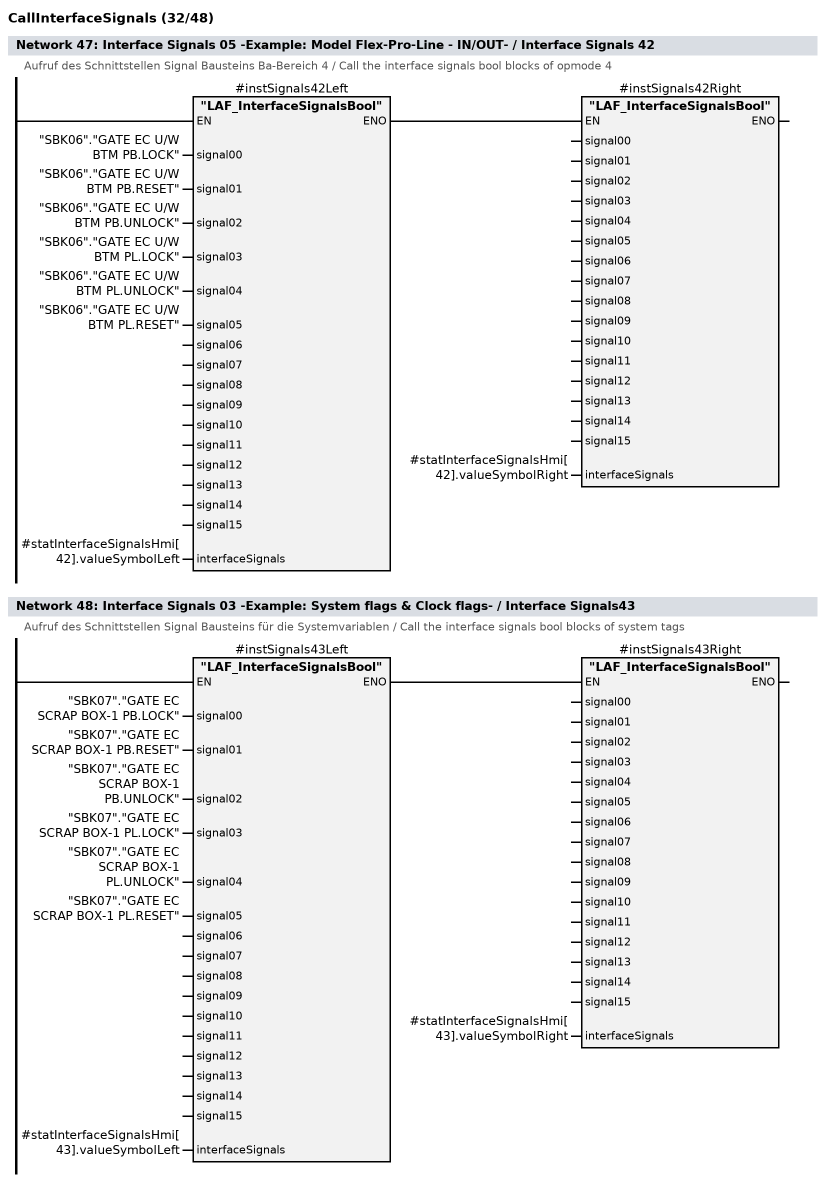
   RUNG wire#powerrail
      #instSignals42Left(signal00 := "SBK06"."GATE EC U/W BTM PB.LOCK", signal01 := "SBK06"."GATE EC U/W BTM PB.RESET", signal02 := "SBK06"."GATE EC U/W BTM PB.UNLOCK", signal03 := "SBK06"."GATE EC U/W BTM PL.LOCK", signal04 := "SBK06"."GATE EC U/W BTM PL.UNLOCK", signal05 := "SBK06"."GATE EC U/W BTM PL.RESET", signal06 :=, signal07 :=, signal08 :=, signal09 :=, signal10 :=, signal11 :=, signal12 :=, signal13 :=, signal14 :=, signal15 :=, interfaceSignals := #statInterfaceSignalsHmi[42].valueSymbolLeft)
      #instSignals42Right(signal00 :=, signal01 :=, signal02 :=, signal03 :=, signal04 :=, signal05 :=, signal06 :=, signal07 :=, signal08 :=, signal09 :=, signal10 :=, signal11 :=, signal12 :=, signal13 :=, signal14 :=, signal15 :=, interfaceSignals := #statInterfaceSignalsHmi[42].valueSymbolRight)
   END_RUNG
   // the same network as SCL:
   #instSignals42Left(signal00 := "SBK06"."GATE EC U/W BTM PB.LOCK",   // "LAF_InterfaceSignalsBool"
                      signal01 := "SBK06"."GATE EC U/W BTM PB.RESET",
                      signal02 := "SBK06"."GATE EC U/W BTM PB.UNLOCK",
                      signal03 := "SBK06"."GATE EC U/W BTM PL.LOCK",
                      signal04 := "SBK06"."GATE EC U/W BTM PL.UNLOCK",
                      signal05 := "SBK06"."GATE EC U/W BTM PL.RESET",
                      interfaceSignals := #statInterfaceSignalsHmi[42].valueSymbolLeft,
                      ENO => #_w1);
   IF #_w1 THEN
       #instSignals42Right(interfaceSignals := #statInterfaceSignalsHmi[42].valueSymbolRight);   // "LAF_InterfaceSignalsBool"
   END_IF;
END_REGION

REGION Network 48: Interface Signals 03 -Example: System flags & Clock flags- / Interface Signals43
   // Aufruf des Schnittstellen Signal Bausteins für die Systemvariablen / Call the interface signals bool blocks of system tags
   RUNG wire#powerrail
      #instSignals43Left(signal00 := "SBK07"."GATE EC SCRAP BOX-1 PB.LOCK", signal01 := "SBK07"."GATE EC SCRAP BOX-1 PB.RESET", signal02 := "SBK07"."GATE EC SCRAP BOX-1 PB.UNLOCK", signal03 := "SBK07"."GATE EC SCRAP BOX-1 PL.LOCK", signal04 := "SBK07"."GATE EC SCRAP BOX-1 PL.UNLOCK", signal05 := "SBK07"."GATE EC SCRAP BOX-1 PL.RESET", signal06 :=, signal07 :=, signal08 :=, signal09 :=, signal10 :=, signal11 :=, signal12 :=, signal13 :=, signal14 :=, signal15 :=, interfaceSignals := #statInterfaceSignalsHmi[43].valueSymbolLeft)
      #instSignals43Right(signal00 :=, signal01 :=, signal02 :=, signal03 :=, signal04 :=, signal05 :=, signal06 :=, signal07 :=, signal08 :=, signal09 :=, signal10 :=, signal11 :=, signal12 :=, signal13 :=, signal14 :=, signal15 :=, interfaceSignals := #statInterfaceSignalsHmi[43].valueSymbolRight)
   END_RUNG
   // the same network as SCL:
   #instSignals43Left(signal00 := "SBK07"."GATE EC SCRAP BOX-1 PB.LOCK",   // "LAF_InterfaceSignalsBool"
                      signal01 := "SBK07"."GATE EC SCRAP BOX-1 PB.RESET",
                      signal02 := "SBK07"."GATE EC SCRAP BOX-1 PB.UNLOCK",
                      signal03 := "SBK07"."GATE EC SCRAP BOX-1 PL.LOCK",
                      signal04 := "SBK07"."GATE EC SCRAP BOX-1 PL.UNLOCK",
                      signal05 := "SBK07"."GATE EC SCRAP BOX-1 PL.RESET",
                      interfaceSignals := #statInterfaceSignalsHmi[43].valueSymbolLeft,
                      ENO => #_w1);
   IF #_w1 THEN
       #instSignals43Right(interfaceSignals := #statInterfaceSignalsHmi[43].valueSymbolRight);   // "LAF_InterfaceSignalsBool"
   END_IF;
END_REGION

REGION Network 49: Interface Signals 04 -Example: Model Flex-Pro-Line - IN/OUT- / Interface Signals 44
   // Aufruf des Schnittstellen Signal Bausteins Ba-Bereich 4 / Call the interface signals bool blocks of opmode 4
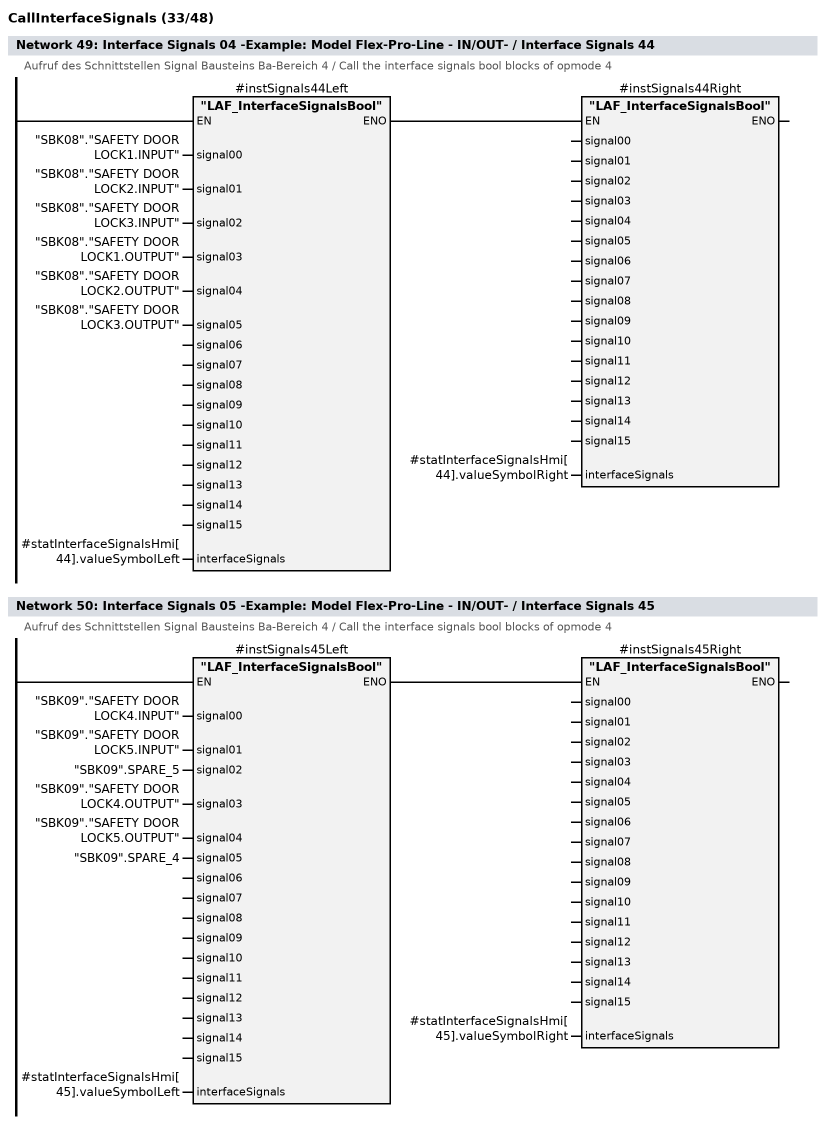
   RUNG wire#powerrail
      #instSignals44Left(signal00 := "SBK08"."SAFETY DOOR LOCK1.INPUT", signal01 := "SBK08"."SAFETY DOOR LOCK2.INPUT", signal02 := "SBK08"."SAFETY DOOR LOCK3.INPUT", signal03 := "SBK08"."SAFETY DOOR LOCK1.OUTPUT", signal04 := "SBK08"."SAFETY DOOR LOCK2.OUTPUT", signal05 := "SBK08"."SAFETY DOOR LOCK3.OUTPUT", signal06 :=, signal07 :=, signal08 :=, signal09 :=, signal10 :=, signal11 :=, signal12 :=, signal13 :=, signal14 :=, signal15 :=, interfaceSignals := #statInterfaceSignalsHmi[44].valueSymbolLeft)
      #instSignals44Right(signal00 :=, signal01 :=, signal02 :=, signal03 :=, signal04 :=, signal05 :=, signal06 :=, signal07 :=, signal08 :=, signal09 :=, signal10 :=, signal11 :=, signal12 :=, signal13 :=, signal14 :=, signal15 :=, interfaceSignals := #statInterfaceSignalsHmi[44].valueSymbolRight)
   END_RUNG
   // the same network as SCL:
   #instSignals44Left(signal00 := "SBK08"."SAFETY DOOR LOCK1.INPUT",   // "LAF_InterfaceSignalsBool"
                      signal01 := "SBK08"."SAFETY DOOR LOCK2.INPUT",
                      signal02 := "SBK08"."SAFETY DOOR LOCK3.INPUT",
                      signal03 := "SBK08"."SAFETY DOOR LOCK1.OUTPUT",
                      signal04 := "SBK08"."SAFETY DOOR LOCK2.OUTPUT",
                      signal05 := "SBK08"."SAFETY DOOR LOCK3.OUTPUT",
                      interfaceSignals := #statInterfaceSignalsHmi[44].valueSymbolLeft,
                      ENO => #_w1);
   IF #_w1 THEN
       #instSignals44Right(interfaceSignals := #statInterfaceSignalsHmi[44].valueSymbolRight);   // "LAF_InterfaceSignalsBool"
   END_IF;
END_REGION

REGION Network 50: Interface Signals 05 -Example: Model Flex-Pro-Line - IN/OUT- / Interface Signals 45
   // Aufruf des Schnittstellen Signal Bausteins Ba-Bereich 4 / Call the interface signals bool blocks of opmode 4
   RUNG wire#powerrail
      #instSignals45Left(signal00 := "SBK09"."SAFETY DOOR LOCK4.INPUT", signal01 := "SBK09"."SAFETY DOOR LOCK5.INPUT", signal02 := "SBK09".SPARE_5, signal03 := "SBK09"."SAFETY DOOR LOCK4.OUTPUT", signal04 := "SBK09"."SAFETY DOOR LOCK5.OUTPUT", signal05 := "SBK09".SPARE_4, signal06 :=, signal07 :=, signal08 :=, signal09 :=, signal10 :=, signal11 :=, signal12 :=, signal13 :=, signal14 :=, signal15 :=, interfaceSignals := #statInterfaceSignalsHmi[45].valueSymbolLeft)
      #instSignals45Right(signal00 :=, signal01 :=, signal02 :=, signal03 :=, signal04 :=, signal05 :=, signal06 :=, signal07 :=, signal08 :=, signal09 :=, signal10 :=, signal11 :=, signal12 :=, signal13 :=, signal14 :=, signal15 :=, interfaceSignals := #statInterfaceSignalsHmi[45].valueSymbolRight)
   END_RUNG
   // the same network as SCL:
   #instSignals45Left(signal00 := "SBK09"."SAFETY DOOR LOCK4.INPUT",   // "LAF_InterfaceSignalsBool"
                      signal01 := "SBK09"."SAFETY DOOR LOCK5.INPUT",
                      signal02 := "SBK09".SPARE_5,
                      signal03 := "SBK09"."SAFETY DOOR LOCK4.OUTPUT",
                      signal04 := "SBK09"."SAFETY DOOR LOCK5.OUTPUT",
                      signal05 := "SBK09".SPARE_4,
                      interfaceSignals := #statInterfaceSignalsHmi[45].valueSymbolLeft,
                      ENO => #_w1);
   IF #_w1 THEN
       #instSignals45Right(interfaceSignals := #statInterfaceSignalsHmi[45].valueSymbolRight);   // "LAF_InterfaceSignalsBool"
   END_IF;
END_REGION

REGION Network 51: Interface Signals 05 -Example: Model Flex-Pro-Line - IN/OUT- / Interface Signals 46
   // Aufruf des Schnittstellen Signal Bausteins Ba-Bereich 4 / Call the interface signals bool blocks of opmode 4
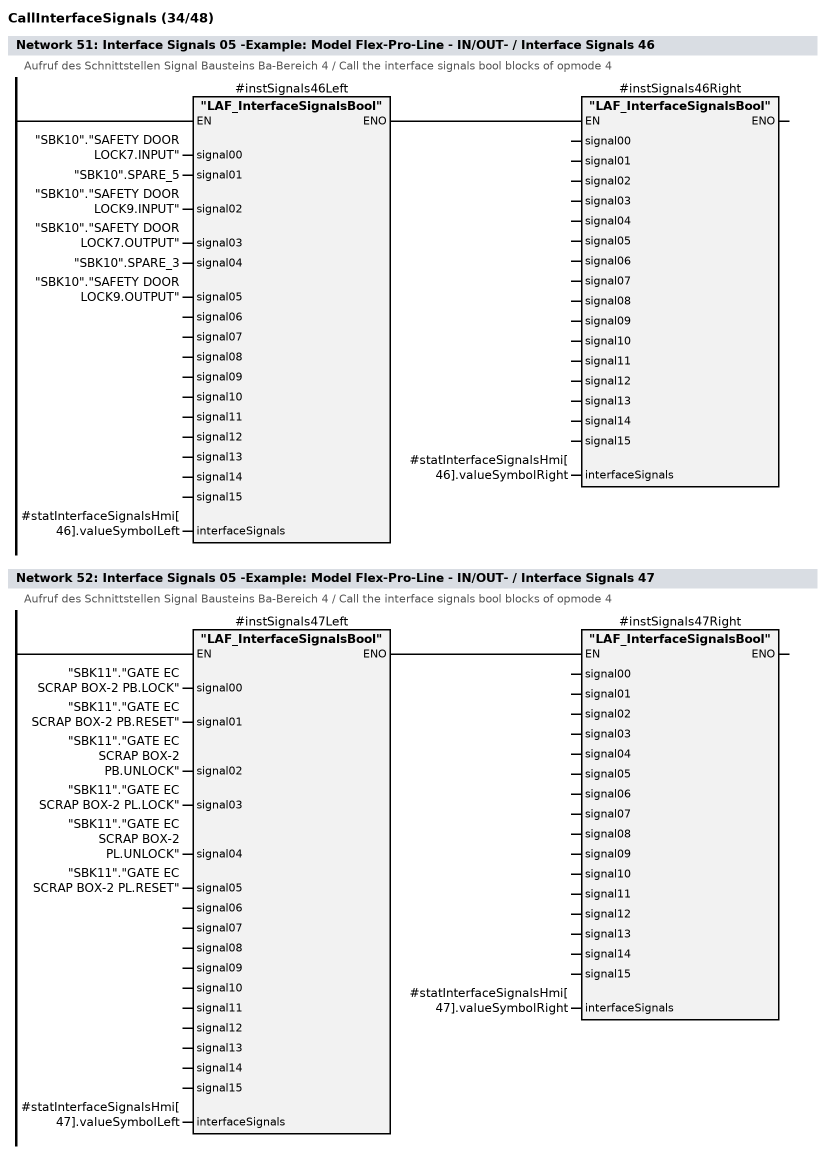
   RUNG wire#powerrail
      #instSignals46Left(signal00 := "SBK10"."SAFETY DOOR LOCK7.INPUT", signal01 := "SBK10".SPARE_5, signal02 := "SBK10"."SAFETY DOOR LOCK9.INPUT", signal03 := "SBK10"."SAFETY DOOR LOCK7.OUTPUT", signal04 := "SBK10".SPARE_3, signal05 := "SBK10"."SAFETY DOOR LOCK9.OUTPUT", signal06 :=, signal07 :=, signal08 :=, signal09 :=, signal10 :=, signal11 :=, signal12 :=, signal13 :=, signal14 :=, signal15 :=, interfaceSignals := #statInterfaceSignalsHmi[46].valueSymbolLeft)
      #instSignals46Right(signal00 :=, signal01 :=, signal02 :=, signal03 :=, signal04 :=, signal05 :=, signal06 :=, signal07 :=, signal08 :=, signal09 :=, signal10 :=, signal11 :=, signal12 :=, signal13 :=, signal14 :=, signal15 :=, interfaceSignals := #statInterfaceSignalsHmi[46].valueSymbolRight)
   END_RUNG
   // the same network as SCL:
   #instSignals46Left(signal00 := "SBK10"."SAFETY DOOR LOCK7.INPUT",   // "LAF_InterfaceSignalsBool"
                      signal01 := "SBK10".SPARE_5,
                      signal02 := "SBK10"."SAFETY DOOR LOCK9.INPUT",
                      signal03 := "SBK10"."SAFETY DOOR LOCK7.OUTPUT",
                      signal04 := "SBK10".SPARE_3,
                      signal05 := "SBK10"."SAFETY DOOR LOCK9.OUTPUT",
                      interfaceSignals := #statInterfaceSignalsHmi[46].valueSymbolLeft,
                      ENO => #_w1);
   IF #_w1 THEN
       #instSignals46Right(interfaceSignals := #statInterfaceSignalsHmi[46].valueSymbolRight);   // "LAF_InterfaceSignalsBool"
   END_IF;
END_REGION

REGION Network 52: Interface Signals 05 -Example: Model Flex-Pro-Line - IN/OUT- / Interface Signals 47
   // Aufruf des Schnittstellen Signal Bausteins Ba-Bereich 4 / Call the interface signals bool blocks of opmode 4
   RUNG wire#powerrail
      #instSignals47Left(signal00 := "SBK11"."GATE EC SCRAP BOX-2 PB.LOCK", signal01 := "SBK11"."GATE EC SCRAP BOX-2 PB.RESET", signal02 := "SBK11"."GATE EC SCRAP BOX-2 PB.UNLOCK", signal03 := "SBK11"."GATE EC SCRAP BOX-2 PL.LOCK", signal04 := "SBK11"."GATE EC SCRAP BOX-2 PL.UNLOCK", signal05 := "SBK11"."GATE EC SCRAP BOX-2 PL.RESET", signal06 :=, signal07 :=, signal08 :=, signal09 :=, signal10 :=, signal11 :=, signal12 :=, signal13 :=, signal14 :=, signal15 :=, interfaceSignals := #statInterfaceSignalsHmi[47].valueSymbolLeft)
      #instSignals47Right(signal00 :=, signal01 :=, signal02 :=, signal03 :=, signal04 :=, signal05 :=, signal06 :=, signal07 :=, signal08 :=, signal09 :=, signal10 :=, signal11 :=, signal12 :=, signal13 :=, signal14 :=, signal15 :=, interfaceSignals := #statInterfaceSignalsHmi[47].valueSymbolRight)
   END_RUNG
   // the same network as SCL:
   #instSignals47Left(signal00 := "SBK11"."GATE EC SCRAP BOX-2 PB.LOCK",   // "LAF_InterfaceSignalsBool"
                      signal01 := "SBK11"."GATE EC SCRAP BOX-2 PB.RESET",
                      signal02 := "SBK11"."GATE EC SCRAP BOX-2 PB.UNLOCK",
                      signal03 := "SBK11"."GATE EC SCRAP BOX-2 PL.LOCK",
                      signal04 := "SBK11"."GATE EC SCRAP BOX-2 PL.UNLOCK",
                      signal05 := "SBK11"."GATE EC SCRAP BOX-2 PL.RESET",
                      interfaceSignals := #statInterfaceSignalsHmi[47].valueSymbolLeft,
                      ENO => #_w1);
   IF #_w1 THEN
       #instSignals47Right(interfaceSignals := #statInterfaceSignalsHmi[47].valueSymbolRight);   // "LAF_InterfaceSignalsBool"
   END_IF;
END_REGION

REGION Network 53: Interface Signals 05 -Example: Model Flex-Pro-Line - IN/OUT- / Interface Signals 48
   // Aufruf des Schnittstellen Signal Bausteins Ba-Bereich 4 / Call the interface signals bool blocks of opmode 4
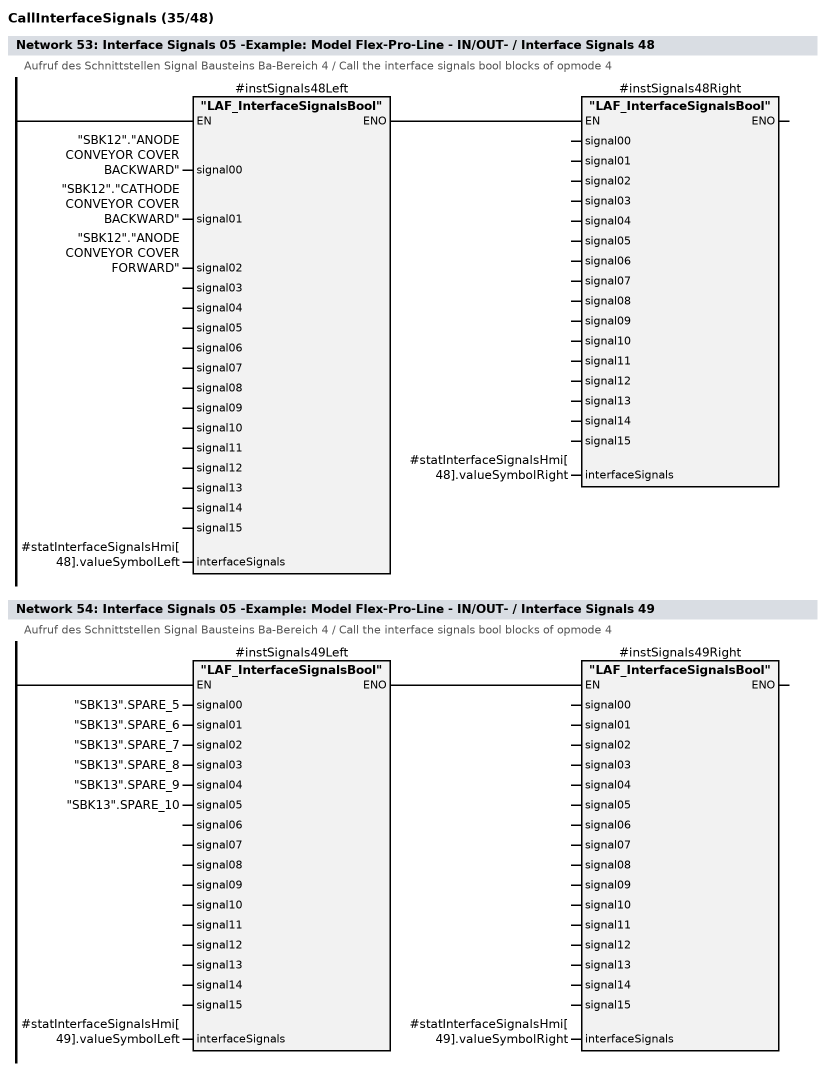
   RUNG wire#powerrail
      #instSignals48Left(signal00 := "SBK12"."ANODE CONVEYOR COVER BACKWARD", signal01 := "SBK12"."CATHODE CONVEYOR COVER BACKWARD", signal02 := "SBK12"."ANODE CONVEYOR COVER FORWARD", signal03 :=, signal04 :=, signal05 :=, signal06 :=, signal07 :=, signal08 :=, signal09 :=, signal10 :=, signal11 :=, signal12 :=, signal13 :=, signal14 :=, signal15 :=, interfaceSignals := #statInterfaceSignalsHmi[48].valueSymbolLeft)
      #instSignals48Right(signal00 :=, signal01 :=, signal02 :=, signal03 :=, signal04 :=, signal05 :=, signal06 :=, signal07 :=, signal08 :=, signal09 :=, signal10 :=, signal11 :=, signal12 :=, signal13 :=, signal14 :=, signal15 :=, interfaceSignals := #statInterfaceSignalsHmi[48].valueSymbolRight)
   END_RUNG
   // the same network as SCL:
   #instSignals48Left(signal00 := "SBK12"."ANODE CONVEYOR COVER BACKWARD",   // "LAF_InterfaceSignalsBool"
                      signal01 := "SBK12"."CATHODE CONVEYOR COVER BACKWARD",
                      signal02 := "SBK12"."ANODE CONVEYOR COVER FORWARD",
                      interfaceSignals := #statInterfaceSignalsHmi[48].valueSymbolLeft,
                      ENO => #_w1);
   IF #_w1 THEN
       #instSignals48Right(interfaceSignals := #statInterfaceSignalsHmi[48].valueSymbolRight);   // "LAF_InterfaceSignalsBool"
   END_IF;
END_REGION

REGION Network 54: Interface Signals 05 -Example: Model Flex-Pro-Line - IN/OUT- / Interface Signals 49
   // Aufruf des Schnittstellen Signal Bausteins Ba-Bereich 4 / Call the interface signals bool blocks of opmode 4
   RUNG wire#powerrail
      #instSignals49Left(signal00 := "SBK13".SPARE_5, signal01 := "SBK13".SPARE_6, signal02 := "SBK13".SPARE_7, signal03 := "SBK13".SPARE_8, signal04 := "SBK13".SPARE_9, signal05 := "SBK13".SPARE_10, signal06 :=, signal07 :=, signal08 :=, signal09 :=, signal10 :=, signal11 :=, signal12 :=, signal13 :=, signal14 :=, signal15 :=, interfaceSignals := #statInterfaceSignalsHmi[49].valueSymbolLeft)
      #instSignals49Right(signal00 :=, signal01 :=, signal02 :=, signal03 :=, signal04 :=, signal05 :=, signal06 :=, signal07 :=, signal08 :=, signal09 :=, signal10 :=, signal11 :=, signal12 :=, signal13 :=, signal14 :=, signal15 :=, interfaceSignals := #statInterfaceSignalsHmi[49].valueSymbolRight)
   END_RUNG
   // the same network as SCL:
   #instSignals49Left(signal00 := "SBK13".SPARE_5,   // "LAF_InterfaceSignalsBool"
                      signal01 := "SBK13".SPARE_6,
                      signal02 := "SBK13".SPARE_7,
                      signal03 := "SBK13".SPARE_8,
                      signal04 := "SBK13".SPARE_9,
                      signal05 := "SBK13".SPARE_10,
                      interfaceSignals := #statInterfaceSignalsHmi[49].valueSymbolLeft,
                      ENO => #_w1);
   IF #_w1 THEN
       #instSignals49Right(interfaceSignals := #statInterfaceSignalsHmi[49].valueSymbolRight);   // "LAF_InterfaceSignalsBool"
   END_IF;
END_REGION

REGION Network 55: Interface Signals 05 -Example: Model Flex-Pro-Line - IN/OUT- / Interface Signals 50
   // Aufruf des Schnittstellen Signal Bausteins Ba-Bereich 4 / Call the interface signals bool blocks of opmode 4
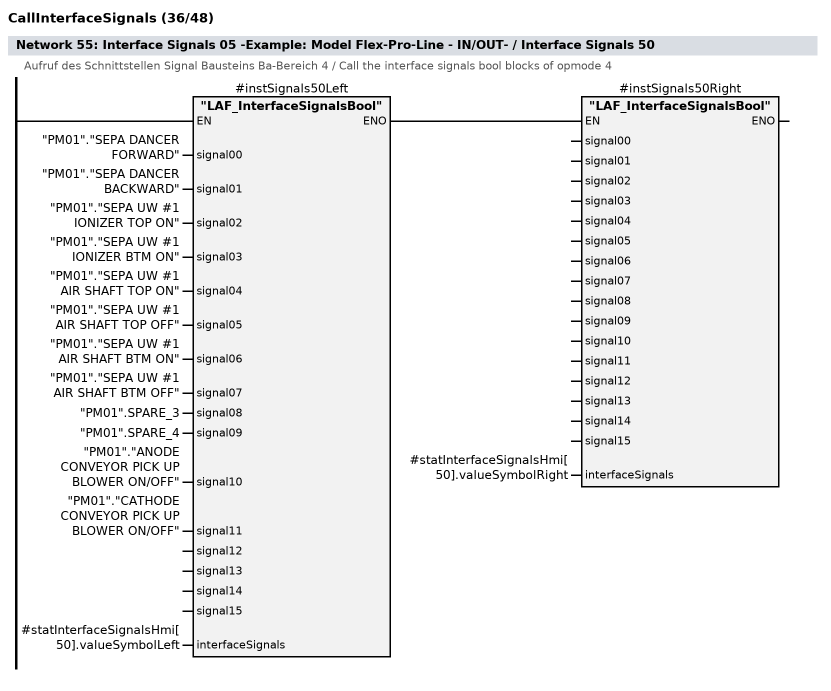
   RUNG wire#powerrail
      #instSignals50Left(signal00 := "PM01"."SEPA DANCER FORWARD", signal01 := "PM01"."SEPA DANCER BACKWARD", signal02 := "PM01"."SEPA UW #1 IONIZER TOP ON", signal03 := "PM01"."SEPA UW #1 IONIZER BTM ON", signal04 := "PM01"."SEPA UW #1 AIR SHAFT TOP ON", signal05 := "PM01"."SEPA UW #1 AIR SHAFT TOP OFF", signal06 := "PM01"."SEPA UW #1 AIR SHAFT BTM ON", signal07 := "PM01"."SEPA UW #1 AIR SHAFT BTM OFF", signal08 := "PM01".SPARE_3, signal09 := "PM01".SPARE_4, signal10 := "PM01"."ANODE CONVEYOR PICK UP BLOWER ON/OFF", signal11 := "PM01"."CATHODE CONVEYOR PICK UP BLOWER ON/OFF", signal12 :=, signal13 :=, signal14 :=, signal15 :=, interfaceSignals := #statInterfaceSignalsHmi[50].valueSymbolLeft)
      #instSignals50Right(signal00 :=, signal01 :=, signal02 :=, signal03 :=, signal04 :=, signal05 :=, signal06 :=, signal07 :=, signal08 :=, signal09 :=, signal10 :=, signal11 :=, signal12 :=, signal13 :=, signal14 :=, signal15 :=, interfaceSignals := #statInterfaceSignalsHmi[50].valueSymbolRight)
   END_RUNG
   // the same network as SCL:
   #instSignals50Left(signal00 := "PM01"."SEPA DANCER FORWARD",   // "LAF_InterfaceSignalsBool"
                      signal01 := "PM01"."SEPA DANCER BACKWARD",
                      signal02 := "PM01"."SEPA UW #1 IONIZER TOP ON",
                      signal03 := "PM01"."SEPA UW #1 IONIZER BTM ON",
                      signal04 := "PM01"."SEPA UW #1 AIR SHAFT TOP ON",
                      signal05 := "PM01"."SEPA UW #1 AIR SHAFT TOP OFF",
                      signal06 := "PM01"."SEPA UW #1 AIR SHAFT BTM ON",
                      signal07 := "PM01"."SEPA UW #1 AIR SHAFT BTM OFF",
                      signal08 := "PM01".SPARE_3,
                      signal09 := "PM01".SPARE_4,
                      signal10 := "PM01"."ANODE CONVEYOR PICK UP BLOWER ON/OFF",
                      signal11 := "PM01"."CATHODE CONVEYOR PICK UP BLOWER ON/OFF",
                      interfaceSignals := #statInterfaceSignalsHmi[50].valueSymbolLeft,
                      ENO => #_w1);
   IF #_w1 THEN
       #instSignals50Right(interfaceSignals := #statInterfaceSignalsHmi[50].valueSymbolRight);   // "LAF_InterfaceSignalsBool"
   END_IF;
END_REGION

REGION Network 56: Interface Signals 05 -Example: Model Flex-Pro-Line - IN/OUT- / Interface Signals 51
   // Aufruf des Schnittstellen Signal Bausteins Ba-Bereich 4 / Call the interface signals bool blocks of opmode 4
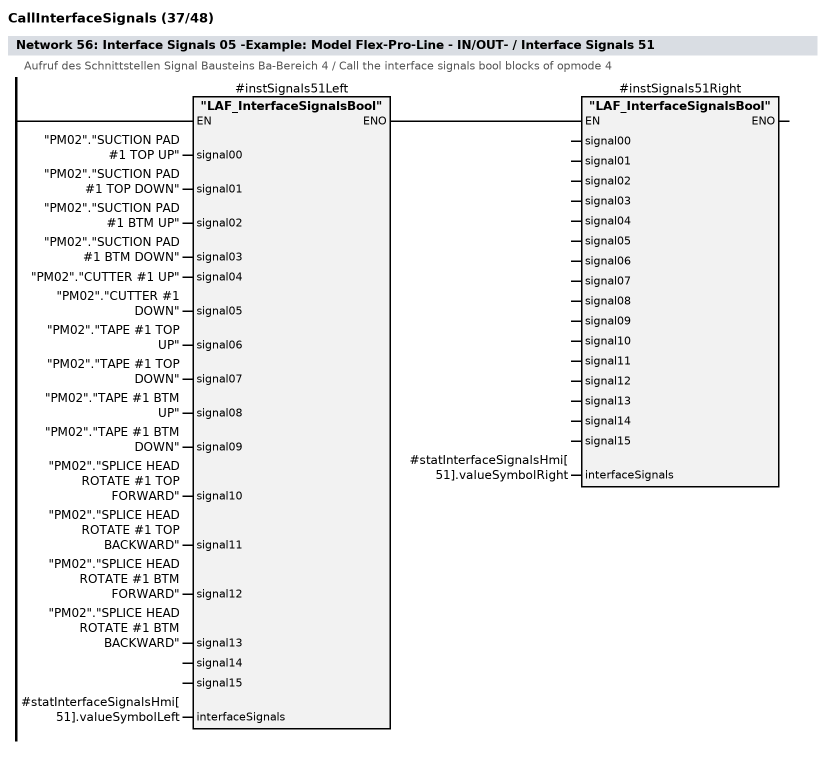
   RUNG wire#powerrail
      #instSignals51Left(signal00 := "PM02"."SUCTION PAD #1 TOP UP", signal01 := "PM02"."SUCTION PAD #1 TOP DOWN", signal02 := "PM02"."SUCTION PAD #1 BTM UP", signal03 := "PM02"."SUCTION PAD #1 BTM DOWN", signal04 := "PM02"."CUTTER #1 UP", signal05 := "PM02"."CUTTER #1 DOWN", signal06 := "PM02"."TAPE #1 TOP UP", signal07 := "PM02"."TAPE #1 TOP DOWN", signal08 := "PM02"."TAPE #1 BTM UP", signal09 := "PM02"."TAPE #1 BTM DOWN", signal10 := "PM02"."SPLICE HEAD ROTATE #1 TOP FORWARD", signal11 := "PM02"."SPLICE HEAD ROTATE #1 TOP BACKWARD", signal12 := "PM02"."SPLICE HEAD ROTATE #1 BTM FORWARD", signal13 := "PM02"."SPLICE HEAD ROTATE #1 BTM BACKWARD", signal14 :=, signal15 :=, interfaceSignals := #statInterfaceSignalsHmi[51].valueSymbolLeft)
      #instSignals51Right(signal00 :=, signal01 :=, signal02 :=, signal03 :=, signal04 :=, signal05 :=, signal06 :=, signal07 :=, signal08 :=, signal09 :=, signal10 :=, signal11 :=, signal12 :=, signal13 :=, signal14 :=, signal15 :=, interfaceSignals := #statInterfaceSignalsHmi[51].valueSymbolRight)
   END_RUNG
   // the same network as SCL:
   #instSignals51Left(signal00 := "PM02"."SUCTION PAD #1 TOP UP",   // "LAF_InterfaceSignalsBool"
                      signal01 := "PM02"."SUCTION PAD #1 TOP DOWN",
                      signal02 := "PM02"."SUCTION PAD #1 BTM UP",
                      signal03 := "PM02"."SUCTION PAD #1 BTM DOWN",
                      signal04 := "PM02"."CUTTER #1 UP",
                      signal05 := "PM02"."CUTTER #1 DOWN",
                      signal06 := "PM02"."TAPE #1 TOP UP",
                      signal07 := "PM02"."TAPE #1 TOP DOWN",
                      signal08 := "PM02"."TAPE #1 BTM UP",
                      signal09 := "PM02"."TAPE #1 BTM DOWN",
                      signal10 := "PM02"."SPLICE HEAD ROTATE #1 TOP FORWARD",
                      signal11 := "PM02"."SPLICE HEAD ROTATE #1 TOP BACKWARD",
                      signal12 := "PM02"."SPLICE HEAD ROTATE #1 BTM FORWARD",
                      signal13 := "PM02"."SPLICE HEAD ROTATE #1 BTM BACKWARD",
                      interfaceSignals := #statInterfaceSignalsHmi[51].valueSymbolLeft,
                      ENO => #_w1);
   IF #_w1 THEN
       #instSignals51Right(interfaceSignals := #statInterfaceSignalsHmi[51].valueSymbolRight);   // "LAF_InterfaceSignalsBool"
   END_IF;
END_REGION

REGION Network 57: Interface Signals 05 -Example: Model Flex-Pro-Line - IN/OUT- / Interface Signals 52
   // Aufruf des Schnittstellen Signal Bausteins Ba-Bereich 4 / Call the interface signals bool blocks of opmode 4
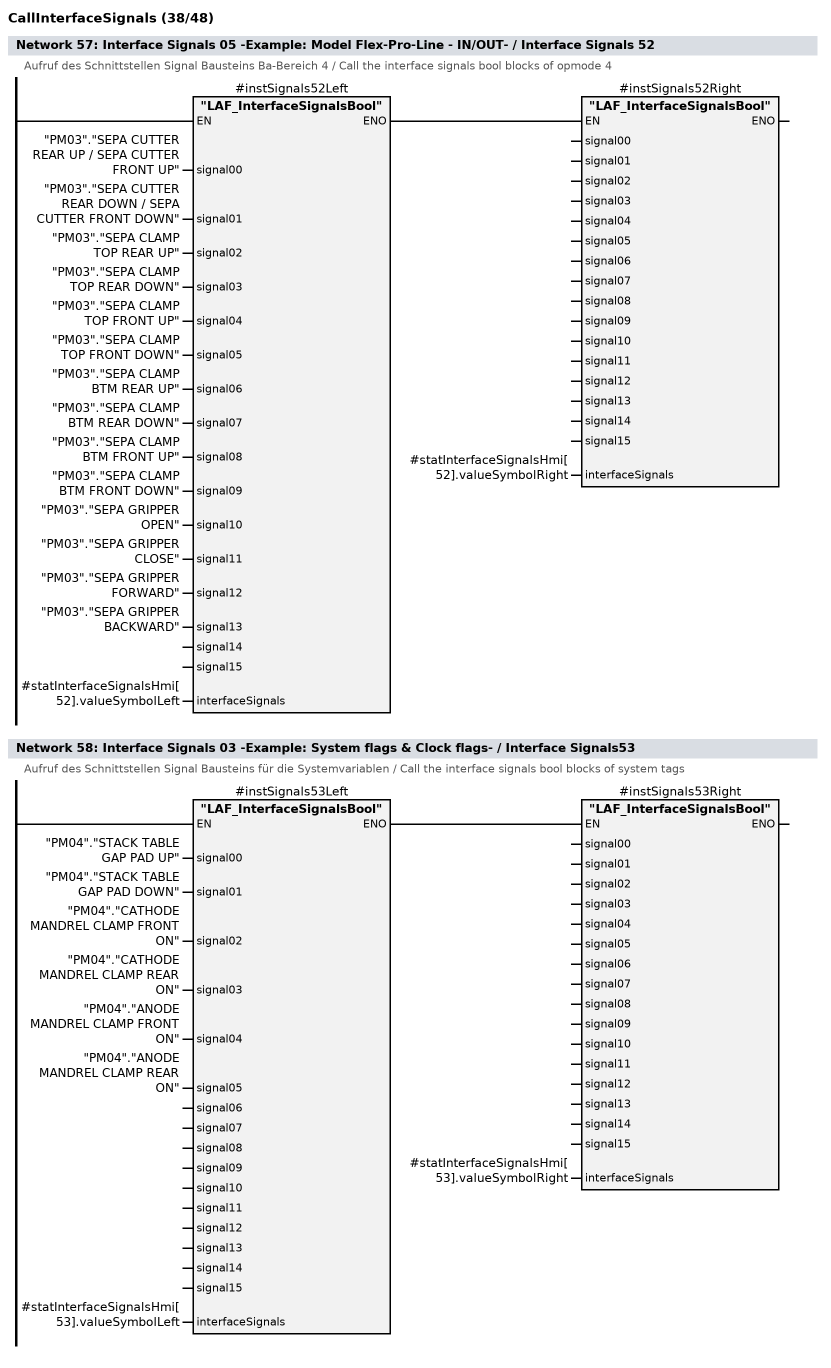
   RUNG wire#powerrail
      #instSignals52Left(signal00 := "PM03"."SEPA CUTTER REAR UP / SEPA CUTTER FRONT UP", signal01 := "PM03"."SEPA CUTTER REAR DOWN / SEPA CUTTER FRONT DOWN", signal02 := "PM03"."SEPA CLAMP TOP REAR UP", signal03 := "PM03"."SEPA CLAMP TOP REAR DOWN", signal04 := "PM03"."SEPA CLAMP TOP FRONT UP", signal05 := "PM03"."SEPA CLAMP TOP FRONT DOWN", signal06 := "PM03"."SEPA CLAMP BTM REAR UP", signal07 := "PM03"."SEPA CLAMP BTM REAR DOWN", signal08 := "PM03"."SEPA CLAMP BTM FRONT UP", signal09 := "PM03"."SEPA CLAMP BTM FRONT DOWN", signal10 := "PM03"."SEPA GRIPPER OPEN", signal11 := "PM03"."SEPA GRIPPER  CLOSE", signal12 := "PM03"."SEPA GRIPPER FORWARD", signal13 := "PM03"."SEPA GRIPPER BACKWARD", signal14 :=, signal15 :=, interfaceSignals := #statInterfaceSignalsHmi[52].valueSymbolLeft)
      #instSignals52Right(signal00 :=, signal01 :=, signal02 :=, signal03 :=, signal04 :=, signal05 :=, signal06 :=, signal07 :=, signal08 :=, signal09 :=, signal10 :=, signal11 :=, signal12 :=, signal13 :=, signal14 :=, signal15 :=, interfaceSignals := #statInterfaceSignalsHmi[52].valueSymbolRight)
   END_RUNG
   // the same network as SCL:
   #instSignals52Left(signal00 := "PM03"."SEPA CUTTER REAR UP / SEPA CUTTER FRONT UP",   // "LAF_InterfaceSignalsBool"
                      signal01 := "PM03"."SEPA CUTTER REAR DOWN / SEPA CUTTER FRONT DOWN",
                      signal02 := "PM03"."SEPA CLAMP TOP REAR UP",
                      signal03 := "PM03"."SEPA CLAMP TOP REAR DOWN",
                      signal04 := "PM03"."SEPA CLAMP TOP FRONT UP",
                      signal05 := "PM03"."SEPA CLAMP TOP FRONT DOWN",
                      signal06 := "PM03"."SEPA CLAMP BTM REAR UP",
                      signal07 := "PM03"."SEPA CLAMP BTM REAR DOWN",
                      signal08 := "PM03"."SEPA CLAMP BTM FRONT UP",
                      signal09 := "PM03"."SEPA CLAMP BTM FRONT DOWN",
                      signal10 := "PM03"."SEPA GRIPPER OPEN",
                      signal11 := "PM03"."SEPA GRIPPER  CLOSE",
                      signal12 := "PM03"."SEPA GRIPPER FORWARD",
                      signal13 := "PM03"."SEPA GRIPPER BACKWARD",
                      interfaceSignals := #statInterfaceSignalsHmi[52].valueSymbolLeft,
                      ENO => #_w1);
   IF #_w1 THEN
       #instSignals52Right(interfaceSignals := #statInterfaceSignalsHmi[52].valueSymbolRight);   // "LAF_InterfaceSignalsBool"
   END_IF;
END_REGION

REGION Network 58: Interface Signals 03 -Example: System flags & Clock flags- / Interface Signals53
   // Aufruf des Schnittstellen Signal Bausteins für die Systemvariablen / Call the interface signals bool blocks of system tags
   RUNG wire#powerrail
      #instSignals53Left(signal00 := "PM04"."STACK TABLE GAP PAD UP", signal01 := "PM04"."STACK TABLE GAP PAD DOWN", signal02 := "PM04"."CATHODE MANDREL CLAMP FRONT ON", signal03 := "PM04"."CATHODE MANDREL CLAMP REAR ON", signal04 := "PM04"."ANODE MANDREL CLAMP FRONT ON", signal05 := "PM04"."ANODE MANDREL CLAMP REAR ON", signal06 :=, signal07 :=, signal08 :=, signal09 :=, signal10 :=, signal11 :=, signal12 :=, signal13 :=, signal14 :=, signal15 :=, interfaceSignals := #statInterfaceSignalsHmi[53].valueSymbolLeft)
      #instSignals53Right(signal00 :=, signal01 :=, signal02 :=, signal03 :=, signal04 :=, signal05 :=, signal06 :=, signal07 :=, signal08 :=, signal09 :=, signal10 :=, signal11 :=, signal12 :=, signal13 :=, signal14 :=, signal15 :=, interfaceSignals := #statInterfaceSignalsHmi[53].valueSymbolRight)
   END_RUNG
   // the same network as SCL:
   #instSignals53Left(signal00 := "PM04"."STACK TABLE GAP PAD UP",   // "LAF_InterfaceSignalsBool"
                      signal01 := "PM04"."STACK TABLE GAP PAD DOWN",
                      signal02 := "PM04"."CATHODE MANDREL CLAMP FRONT ON",
                      signal03 := "PM04"."CATHODE MANDREL CLAMP REAR ON",
                      signal04 := "PM04"."ANODE MANDREL CLAMP FRONT ON",
                      signal05 := "PM04"."ANODE MANDREL CLAMP REAR ON",
                      interfaceSignals := #statInterfaceSignalsHmi[53].valueSymbolLeft,
                      ENO => #_w1);
   IF #_w1 THEN
       #instSignals53Right(interfaceSignals := #statInterfaceSignalsHmi[53].valueSymbolRight);   // "LAF_InterfaceSignalsBool"
   END_IF;
END_REGION

REGION Network 59: Interface Signals 04 -Example: Model Flex-Pro-Line - IN/OUT- / Interface Signals 54
   // Aufruf des Schnittstellen Signal Bausteins Ba-Bereich 4 / Call the interface signals bool blocks of opmode 4
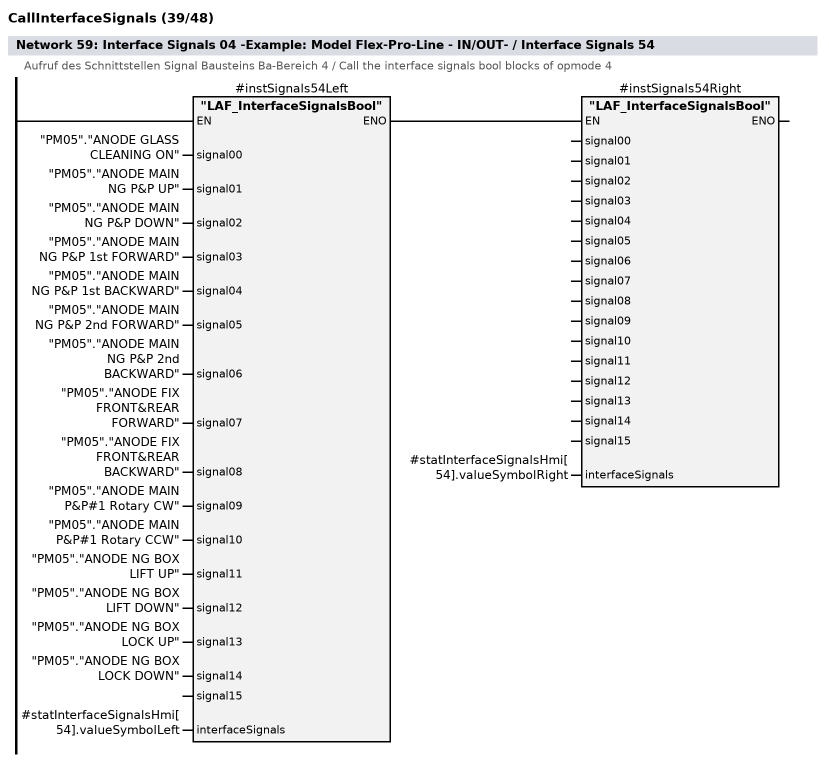
   RUNG wire#powerrail
      #instSignals54Left(signal00 := "PM05"."ANODE GLASS CLEANING ON", signal01 := "PM05"."ANODE MAIN NG P&P UP", signal02 := "PM05"."ANODE MAIN NG P&P DOWN", signal03 := "PM05"."ANODE MAIN NG P&P 1st FORWARD", signal04 := "PM05"."ANODE MAIN NG P&P 1st BACKWARD", signal05 := "PM05"."ANODE MAIN NG P&P 2nd FORWARD", signal06 := "PM05"."ANODE MAIN NG P&P 2nd BACKWARD", signal07 := "PM05"."ANODE FIX FRONT&REAR FORWARD", signal08 := "PM05"."ANODE FIX FRONT&REAR BACKWARD", signal09 := "PM05"."ANODE MAIN P&P#1 Rotary CW", signal10 := "PM05"."ANODE MAIN P&P#1 Rotary CCW", signal11 := "PM05"."ANODE NG BOX LIFT UP", signal12 := "PM05"."ANODE NG BOX LIFT DOWN", signal13 := "PM05"."ANODE NG BOX LOCK UP", signal14 := "PM05"."ANODE NG BOX LOCK DOWN", signal15 :=, interfaceSignals := #statInterfaceSignalsHmi[54].valueSymbolLeft)
      #instSignals54Right(signal00 :=, signal01 :=, signal02 :=, signal03 :=, signal04 :=, signal05 :=, signal06 :=, signal07 :=, signal08 :=, signal09 :=, signal10 :=, signal11 :=, signal12 :=, signal13 :=, signal14 :=, signal15 :=, interfaceSignals := #statInterfaceSignalsHmi[54].valueSymbolRight)
   END_RUNG
   // the same network as SCL:
   #instSignals54Left(signal00 := "PM05"."ANODE GLASS CLEANING ON",   // "LAF_InterfaceSignalsBool"
                      signal01 := "PM05"."ANODE MAIN NG P&P UP",
                      signal02 := "PM05"."ANODE MAIN NG P&P DOWN",
                      signal03 := "PM05"."ANODE MAIN NG P&P 1st FORWARD",
                      signal04 := "PM05"."ANODE MAIN NG P&P 1st BACKWARD",
                      signal05 := "PM05"."ANODE MAIN NG P&P 2nd FORWARD",
                      signal06 := "PM05"."ANODE MAIN NG P&P 2nd BACKWARD",
                      signal07 := "PM05"."ANODE FIX FRONT&REAR FORWARD",
                      signal08 := "PM05"."ANODE FIX FRONT&REAR BACKWARD",
                      signal09 := "PM05"."ANODE MAIN P&P#1 Rotary CW",
                      signal10 := "PM05"."ANODE MAIN P&P#1 Rotary CCW",
                      signal11 := "PM05"."ANODE NG BOX LIFT UP",
                      signal12 := "PM05"."ANODE NG BOX LIFT DOWN",
                      signal13 := "PM05"."ANODE NG BOX LOCK UP",
                      signal14 := "PM05"."ANODE NG BOX LOCK DOWN",
                      interfaceSignals := #statInterfaceSignalsHmi[54].valueSymbolLeft,
                      ENO => #_w1);
   IF #_w1 THEN
       #instSignals54Right(interfaceSignals := #statInterfaceSignalsHmi[54].valueSymbolRight);   // "LAF_InterfaceSignalsBool"
   END_IF;
END_REGION

REGION Network 60: Interface Signals 05 -Example: Model Flex-Pro-Line - IN/OUT- / Interface Signals 55
   // Aufruf des Schnittstellen Signal Bausteins Ba-Bereich 4 / Call the interface signals bool blocks of opmode 4
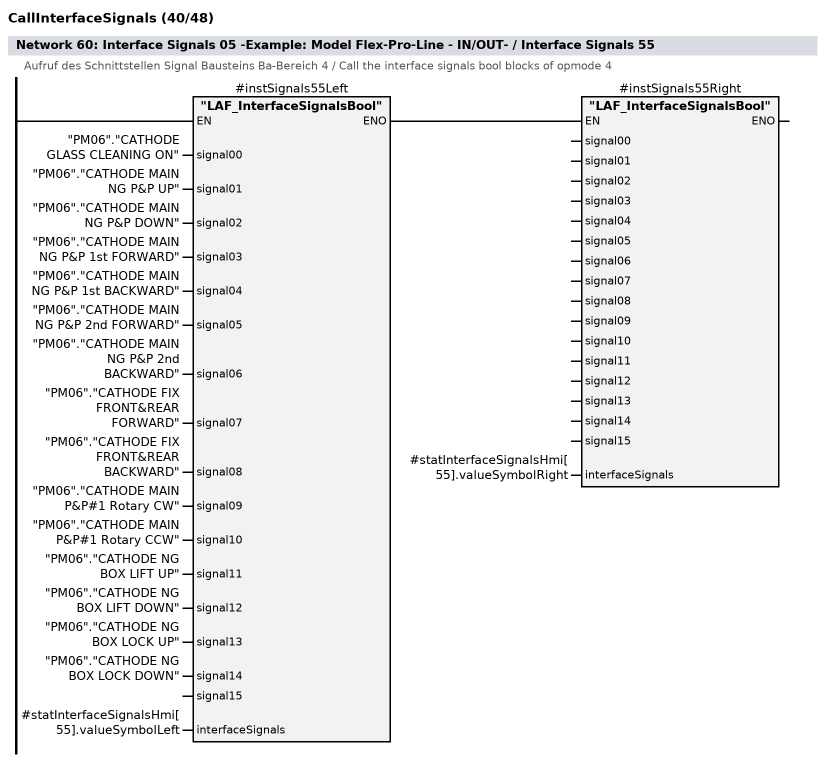
   RUNG wire#powerrail
      #instSignals55Left(signal00 := "PM06"."CATHODE GLASS CLEANING ON", signal01 := "PM06"."CATHODE MAIN NG P&P UP", signal02 := "PM06"."CATHODE MAIN NG P&P DOWN", signal03 := "PM06"."CATHODE MAIN NG P&P 1st FORWARD", signal04 := "PM06"."CATHODE MAIN NG P&P 1st BACKWARD", signal05 := "PM06"."CATHODE MAIN NG P&P 2nd FORWARD", signal06 := "PM06"."CATHODE MAIN NG P&P 2nd BACKWARD", signal07 := "PM06"."CATHODE FIX FRONT&REAR FORWARD", signal08 := "PM06"."CATHODE FIX FRONT&REAR BACKWARD", signal09 := "PM06"."CATHODE MAIN P&P#1 Rotary CW", signal10 := "PM06"."CATHODE MAIN P&P#1 Rotary CCW", signal11 := "PM06"."CATHODE NG BOX LIFT UP", signal12 := "PM06"."CATHODE NG BOX LIFT DOWN", signal13 := "PM06"."CATHODE NG BOX LOCK UP", signal14 := "PM06"."CATHODE NG BOX LOCK DOWN", signal15 :=, interfaceSignals := #statInterfaceSignalsHmi[55].valueSymbolLeft)
      #instSignals55Right(signal00 :=, signal01 :=, signal02 :=, signal03 :=, signal04 :=, signal05 :=, signal06 :=, signal07 :=, signal08 :=, signal09 :=, signal10 :=, signal11 :=, signal12 :=, signal13 :=, signal14 :=, signal15 :=, interfaceSignals := #statInterfaceSignalsHmi[55].valueSymbolRight)
   END_RUNG
   // the same network as SCL:
   #instSignals55Left(signal00 := "PM06"."CATHODE GLASS CLEANING ON",   // "LAF_InterfaceSignalsBool"
                      signal01 := "PM06"."CATHODE MAIN NG P&P UP",
                      signal02 := "PM06"."CATHODE MAIN NG P&P DOWN",
                      signal03 := "PM06"."CATHODE MAIN NG P&P 1st FORWARD",
                      signal04 := "PM06"."CATHODE MAIN NG P&P 1st BACKWARD",
                      signal05 := "PM06"."CATHODE MAIN NG P&P 2nd FORWARD",
                      signal06 := "PM06"."CATHODE MAIN NG P&P 2nd BACKWARD",
                      signal07 := "PM06"."CATHODE FIX FRONT&REAR FORWARD",
                      signal08 := "PM06"."CATHODE FIX FRONT&REAR BACKWARD",
                      signal09 := "PM06"."CATHODE MAIN P&P#1 Rotary CW",
                      signal10 := "PM06"."CATHODE MAIN P&P#1 Rotary CCW",
                      signal11 := "PM06"."CATHODE NG BOX LIFT UP",
                      signal12 := "PM06"."CATHODE NG BOX LIFT DOWN",
                      signal13 := "PM06"."CATHODE NG BOX LOCK UP",
                      signal14 := "PM06"."CATHODE NG BOX LOCK DOWN",
                      interfaceSignals := #statInterfaceSignalsHmi[55].valueSymbolLeft,
                      ENO => #_w1);
   IF #_w1 THEN
       #instSignals55Right(interfaceSignals := #statInterfaceSignalsHmi[55].valueSymbolRight);   // "LAF_InterfaceSignalsBool"
   END_IF;
END_REGION

REGION Network 61: Interface Signals 05 -Example: Model Flex-Pro-Line - IN/OUT- / Interface Signals 56
   // Aufruf des Schnittstellen Signal Bausteins Ba-Bereich 4 / Call the interface signals bool blocks of opmode 4
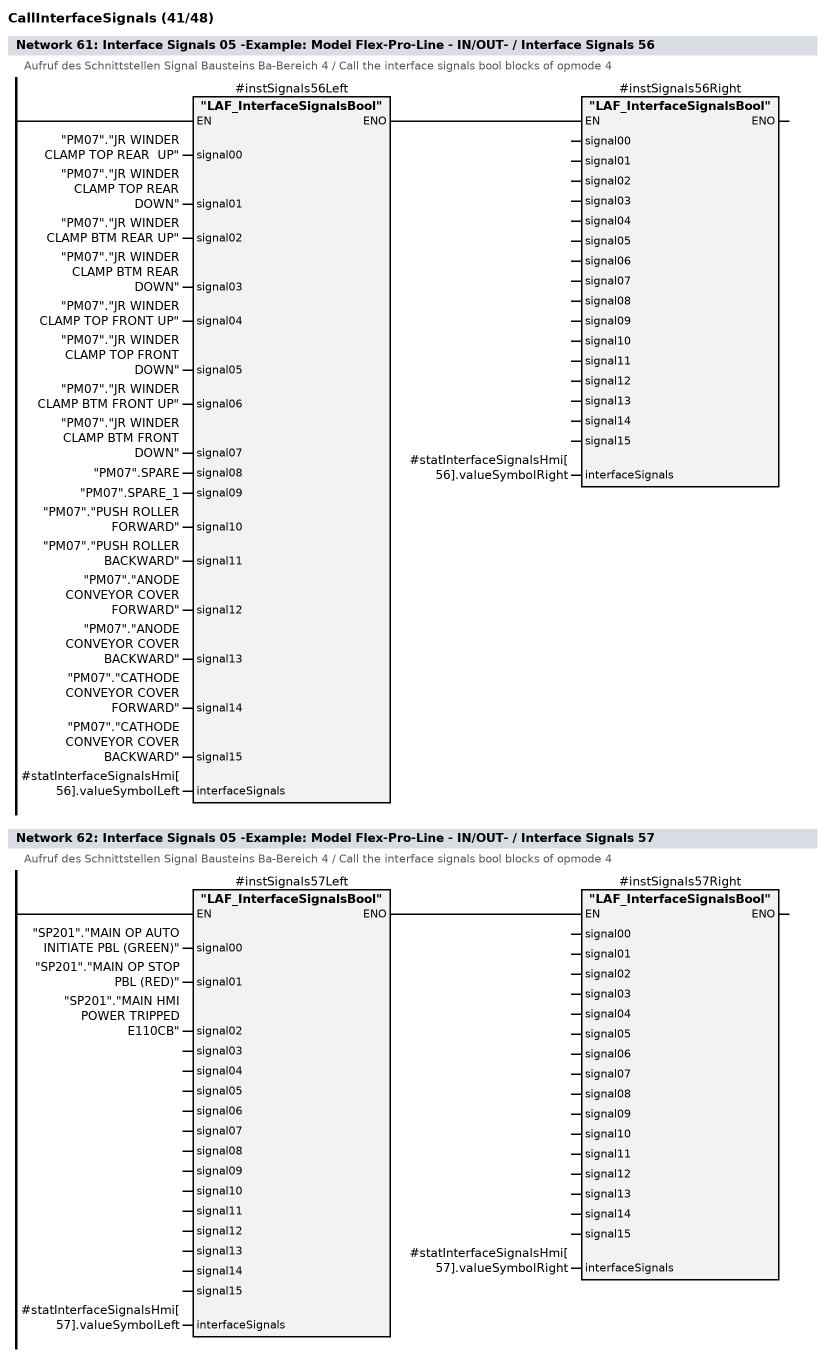
   RUNG wire#powerrail
      #instSignals56Left(signal00 := "PM07"."JR WINDER CLAMP TOP REAR  UP", signal01 := "PM07"."JR WINDER CLAMP TOP REAR  DOWN", signal02 := "PM07"."JR WINDER CLAMP BTM REAR UP", signal03 := "PM07"."JR WINDER CLAMP BTM REAR DOWN", signal04 := "PM07"."JR WINDER CLAMP TOP FRONT UP", signal05 := "PM07"."JR WINDER CLAMP TOP FRONT DOWN", signal06 := "PM07"."JR WINDER CLAMP BTM FRONT UP", signal07 := "PM07"."JR WINDER CLAMP BTM FRONT DOWN", signal08 := "PM07".SPARE, signal09 := "PM07".SPARE_1, signal10 := "PM07"."PUSH ROLLER FORWARD", signal11 := "PM07"."PUSH ROLLER BACKWARD", signal12 := "PM07"."ANODE CONVEYOR COVER FORWARD", signal13 := "PM07"."ANODE CONVEYOR COVER BACKWARD", signal14 := "PM07"."CATHODE CONVEYOR COVER FORWARD", signal15 := "PM07"."CATHODE CONVEYOR COVER BACKWARD", interfaceSignals := #statInterfaceSignalsHmi[56].valueSymbolLeft)
      #instSignals56Right(signal00 :=, signal01 :=, signal02 :=, signal03 :=, signal04 :=, signal05 :=, signal06 :=, signal07 :=, signal08 :=, signal09 :=, signal10 :=, signal11 :=, signal12 :=, signal13 :=, signal14 :=, signal15 :=, interfaceSignals := #statInterfaceSignalsHmi[56].valueSymbolRight)
   END_RUNG
   // the same network as SCL:
   #instSignals56Left(signal00 := "PM07"."JR WINDER CLAMP TOP REAR  UP",   // "LAF_InterfaceSignalsBool"
                      signal01 := "PM07"."JR WINDER CLAMP TOP REAR  DOWN",
                      signal02 := "PM07"."JR WINDER CLAMP BTM REAR UP",
                      signal03 := "PM07"."JR WINDER CLAMP BTM REAR DOWN",
                      signal04 := "PM07"."JR WINDER CLAMP TOP FRONT UP",
                      signal05 := "PM07"."JR WINDER CLAMP TOP FRONT DOWN",
                      signal06 := "PM07"."JR WINDER CLAMP BTM FRONT UP",
                      signal07 := "PM07"."JR WINDER CLAMP BTM FRONT DOWN",
                      signal08 := "PM07".SPARE,
                      signal09 := "PM07".SPARE_1,
                      signal10 := "PM07"."PUSH ROLLER FORWARD",
                      signal11 := "PM07"."PUSH ROLLER BACKWARD",
                      signal12 := "PM07"."ANODE CONVEYOR COVER FORWARD",
                      signal13 := "PM07"."ANODE CONVEYOR COVER BACKWARD",
                      signal14 := "PM07"."CATHODE CONVEYOR COVER FORWARD",
                      signal15 := "PM07"."CATHODE CONVEYOR COVER BACKWARD",
                      interfaceSignals := #statInterfaceSignalsHmi[56].valueSymbolLeft,
                      ENO => #_w1);
   IF #_w1 THEN
       #instSignals56Right(interfaceSignals := #statInterfaceSignalsHmi[56].valueSymbolRight);   // "LAF_InterfaceSignalsBool"
   END_IF;
END_REGION

REGION Network 62: Interface Signals 05 -Example: Model Flex-Pro-Line - IN/OUT- / Interface Signals 57
   // Aufruf des Schnittstellen Signal Bausteins Ba-Bereich 4 / Call the interface signals bool blocks of opmode 4
   RUNG wire#powerrail
      #instSignals57Left(signal00 := "SP201"."MAIN OP AUTO INITIATE PBL (GREEN)", signal01 := "SP201"."MAIN OP STOP PBL (RED)", signal02 := "SP201"."MAIN HMI POWER TRIPPED E110CB", signal03 :=, signal04 :=, signal05 :=, signal06 :=, signal07 :=, signal08 :=, signal09 :=, signal10 :=, signal11 :=, signal12 :=, signal13 :=, signal14 :=, signal15 :=, interfaceSignals := #statInterfaceSignalsHmi[57].valueSymbolLeft)
      #instSignals57Right(signal00 :=, signal01 :=, signal02 :=, signal03 :=, signal04 :=, signal05 :=, signal06 :=, signal07 :=, signal08 :=, signal09 :=, signal10 :=, signal11 :=, signal12 :=, signal13 :=, signal14 :=, signal15 :=, interfaceSignals := #statInterfaceSignalsHmi[57].valueSymbolRight)
   END_RUNG
   // the same network as SCL:
   #instSignals57Left(signal00 := "SP201"."MAIN OP AUTO INITIATE PBL (GREEN)",   // "LAF_InterfaceSignalsBool"
                      signal01 := "SP201"."MAIN OP STOP PBL (RED)",
                      signal02 := "SP201"."MAIN HMI POWER TRIPPED E110CB",
                      interfaceSignals := #statInterfaceSignalsHmi[57].valueSymbolLeft,
                      ENO => #_w1);
   IF #_w1 THEN
       #instSignals57Right(interfaceSignals := #statInterfaceSignalsHmi[57].valueSymbolRight);   // "LAF_InterfaceSignalsBool"
   END_IF;
END_REGION

REGION Network 63: Interface Signals 05 -Example: Model Flex-Pro-Line - IN/OUT- / Interface Signals 58
   // Aufruf des Schnittstellen Signal Bausteins Ba-Bereich 4 / Call the interface signals bool blocks of opmode 4
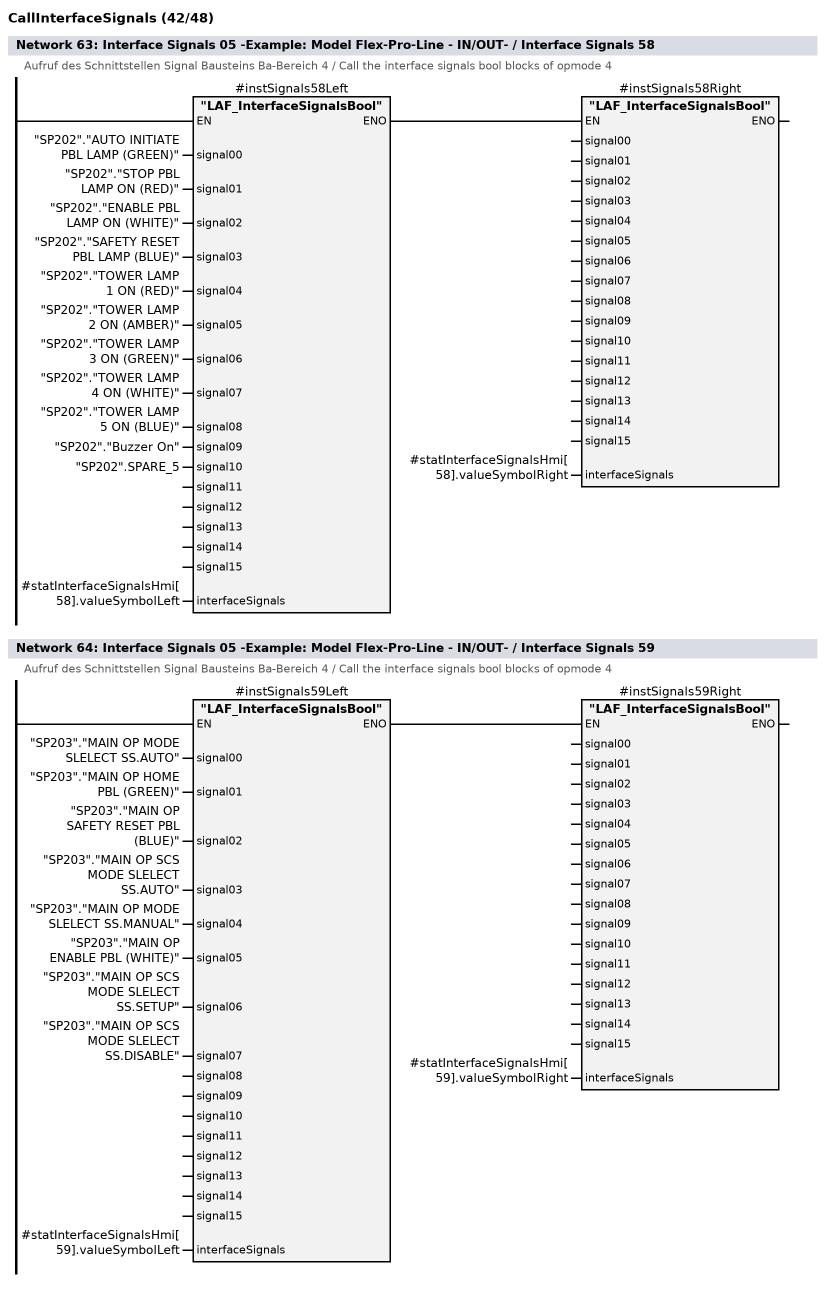
   RUNG wire#powerrail
      #instSignals58Left(signal00 := "SP202"."AUTO INITIATE PBL LAMP (GREEN)", signal01 := "SP202"."STOP PBL LAMP ON (RED)", signal02 := "SP202"."ENABLE PBL LAMP ON (WHITE)", signal03 := "SP202"."SAFETY RESET PBL LAMP (BLUE)", signal04 := "SP202"."TOWER LAMP 1 ON (RED)", signal05 := "SP202"."TOWER LAMP 2 ON (AMBER)", signal06 := "SP202"."TOWER LAMP 3 ON (GREEN)", signal07 := "SP202"."TOWER LAMP 4 ON (WHITE)", signal08 := "SP202"."TOWER LAMP 5 ON (BLUE)", signal09 := "SP202"."Buzzer On", signal10 := "SP202".SPARE_5, signal11 :=, signal12 :=, signal13 :=, signal14 :=, signal15 :=, interfaceSignals := #statInterfaceSignalsHmi[58].valueSymbolLeft)
      #instSignals58Right(signal00 :=, signal01 :=, signal02 :=, signal03 :=, signal04 :=, signal05 :=, signal06 :=, signal07 :=, signal08 :=, signal09 :=, signal10 :=, signal11 :=, signal12 :=, signal13 :=, signal14 :=, signal15 :=, interfaceSignals := #statInterfaceSignalsHmi[58].valueSymbolRight)
   END_RUNG
   // the same network as SCL:
   #instSignals58Left(signal00 := "SP202"."AUTO INITIATE PBL LAMP (GREEN)",   // "LAF_InterfaceSignalsBool"
                      signal01 := "SP202"."STOP PBL LAMP ON (RED)",
                      signal02 := "SP202"."ENABLE PBL LAMP ON (WHITE)",
                      signal03 := "SP202"."SAFETY RESET PBL LAMP (BLUE)",
                      signal04 := "SP202"."TOWER LAMP 1 ON (RED)",
                      signal05 := "SP202"."TOWER LAMP 2 ON (AMBER)",
                      signal06 := "SP202"."TOWER LAMP 3 ON (GREEN)",
                      signal07 := "SP202"."TOWER LAMP 4 ON (WHITE)",
                      signal08 := "SP202"."TOWER LAMP 5 ON (BLUE)",
                      signal09 := "SP202"."Buzzer On",
                      signal10 := "SP202".SPARE_5,
                      interfaceSignals := #statInterfaceSignalsHmi[58].valueSymbolLeft,
                      ENO => #_w1);
   IF #_w1 THEN
       #instSignals58Right(interfaceSignals := #statInterfaceSignalsHmi[58].valueSymbolRight);   // "LAF_InterfaceSignalsBool"
   END_IF;
END_REGION

REGION Network 64: Interface Signals 05 -Example: Model Flex-Pro-Line - IN/OUT- / Interface Signals 59
   // Aufruf des Schnittstellen Signal Bausteins Ba-Bereich 4 / Call the interface signals bool blocks of opmode 4
   RUNG wire#powerrail
      #instSignals59Left(signal00 := "SP203"."MAIN OP MODE SLELECT SS.AUTO", signal01 := "SP203"."MAIN OP HOME PBL (GREEN)", signal02 := "SP203"."MAIN OP SAFETY RESET PBL (BLUE)", signal03 := "SP203"."MAIN OP SCS MODE SLELECT SS.AUTO", signal04 := "SP203"."MAIN OP MODE SLELECT SS.MANUAL", signal05 := "SP203"."MAIN OP ENABLE PBL (WHITE)", signal06 := "SP203"."MAIN OP SCS MODE SLELECT SS.SETUP", signal07 := "SP203"."MAIN OP SCS MODE SLELECT SS.DISABLE", signal08 :=, signal09 :=, signal10 :=, signal11 :=, signal12 :=, signal13 :=, signal14 :=, signal15 :=, interfaceSignals := #statInterfaceSignalsHmi[59].valueSymbolLeft)
      #instSignals59Right(signal00 :=, signal01 :=, signal02 :=, signal03 :=, signal04 :=, signal05 :=, signal06 :=, signal07 :=, signal08 :=, signal09 :=, signal10 :=, signal11 :=, signal12 :=, signal13 :=, signal14 :=, signal15 :=, interfaceSignals := #statInterfaceSignalsHmi[59].valueSymbolRight)
   END_RUNG
   // the same network as SCL:
   #instSignals59Left(signal00 := "SP203"."MAIN OP MODE SLELECT SS.AUTO",   // "LAF_InterfaceSignalsBool"
                      signal01 := "SP203"."MAIN OP HOME PBL (GREEN)",
                      signal02 := "SP203"."MAIN OP SAFETY RESET PBL (BLUE)",
                      signal03 := "SP203"."MAIN OP SCS MODE SLELECT SS.AUTO",
                      signal04 := "SP203"."MAIN OP MODE SLELECT SS.MANUAL",
                      signal05 := "SP203"."MAIN OP ENABLE PBL (WHITE)",
                      signal06 := "SP203"."MAIN OP SCS MODE SLELECT SS.SETUP",
                      signal07 := "SP203"."MAIN OP SCS MODE SLELECT SS.DISABLE",
                      interfaceSignals := #statInterfaceSignalsHmi[59].valueSymbolLeft,
                      ENO => #_w1);
   IF #_w1 THEN
       #instSignals59Right(interfaceSignals := #statInterfaceSignalsHmi[59].valueSymbolRight);   // "LAF_InterfaceSignalsBool"
   END_IF;
END_REGION

REGION Network 65: Interface Signals 05 -Example: Model Flex-Pro-Line - IN/OUT- / Interface Signals 60
   // Aufruf des Schnittstellen Signal Bausteins Ba-Bereich 4 / Call the interface signals bool blocks of opmode 4
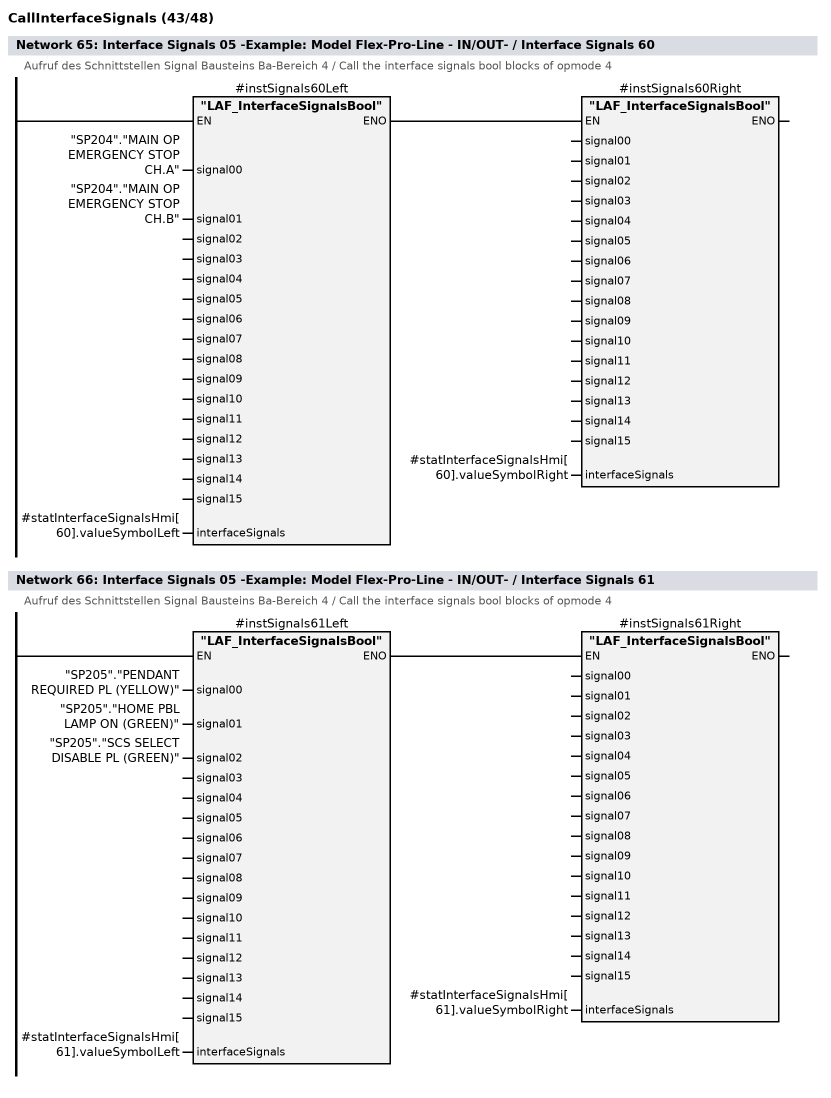
   RUNG wire#powerrail
      #instSignals60Left(signal00 := "SP204"."MAIN OP EMERGENCY STOP CH.A", signal01 := "SP204"."MAIN OP EMERGENCY STOP CH.B", signal02 :=, signal03 :=, signal04 :=, signal05 :=, signal06 :=, signal07 :=, signal08 :=, signal09 :=, signal10 :=, signal11 :=, signal12 :=, signal13 :=, signal14 :=, signal15 :=, interfaceSignals := #statInterfaceSignalsHmi[60].valueSymbolLeft)
      #instSignals60Right(signal00 :=, signal01 :=, signal02 :=, signal03 :=, signal04 :=, signal05 :=, signal06 :=, signal07 :=, signal08 :=, signal09 :=, signal10 :=, signal11 :=, signal12 :=, signal13 :=, signal14 :=, signal15 :=, interfaceSignals := #statInterfaceSignalsHmi[60].valueSymbolRight)
   END_RUNG
   // the same network as SCL:
   #instSignals60Left(signal00 := "SP204"."MAIN OP EMERGENCY STOP CH.A",   // "LAF_InterfaceSignalsBool"
                      signal01 := "SP204"."MAIN OP EMERGENCY STOP CH.B",
                      interfaceSignals := #statInterfaceSignalsHmi[60].valueSymbolLeft,
                      ENO => #_w1);
   IF #_w1 THEN
       #instSignals60Right(interfaceSignals := #statInterfaceSignalsHmi[60].valueSymbolRight);   // "LAF_InterfaceSignalsBool"
   END_IF;
END_REGION

REGION Network 66: Interface Signals 05 -Example: Model Flex-Pro-Line - IN/OUT- / Interface Signals 61
   // Aufruf des Schnittstellen Signal Bausteins Ba-Bereich 4 / Call the interface signals bool blocks of opmode 4
   RUNG wire#powerrail
      #instSignals61Left(signal00 := "SP205"."PENDANT REQUIRED PL (YELLOW)", signal01 := "SP205"."HOME PBL LAMP ON (GREEN)", signal02 := "SP205"."SCS SELECT DISABLE PL (GREEN)", signal03 :=, signal04 :=, signal05 :=, signal06 :=, signal07 :=, signal08 :=, signal09 :=, signal10 :=, signal11 :=, signal12 :=, signal13 :=, signal14 :=, signal15 :=, interfaceSignals := #statInterfaceSignalsHmi[61].valueSymbolLeft)
      #instSignals61Right(signal00 :=, signal01 :=, signal02 :=, signal03 :=, signal04 :=, signal05 :=, signal06 :=, signal07 :=, signal08 :=, signal09 :=, signal10 :=, signal11 :=, signal12 :=, signal13 :=, signal14 :=, signal15 :=, interfaceSignals := #statInterfaceSignalsHmi[61].valueSymbolRight)
   END_RUNG
   // the same network as SCL:
   #instSignals61Left(signal00 := "SP205"."PENDANT REQUIRED PL (YELLOW)",   // "LAF_InterfaceSignalsBool"
                      signal01 := "SP205"."HOME PBL LAMP ON (GREEN)",
                      signal02 := "SP205"."SCS SELECT DISABLE PL (GREEN)",
                      interfaceSignals := #statInterfaceSignalsHmi[61].valueSymbolLeft,
                      ENO => #_w1);
   IF #_w1 THEN
       #instSignals61Right(interfaceSignals := #statInterfaceSignalsHmi[61].valueSymbolRight);   // "LAF_InterfaceSignalsBool"
   END_IF;
END_REGION

REGION Network 67: Interface Signals 05 -Example: Model Flex-Pro-Line - IN/OUT- / Interface Signals 62
   // Aufruf des Schnittstellen Signal Bausteins Ba-Bereich 4 / Call the interface signals bool blocks of opmode 4
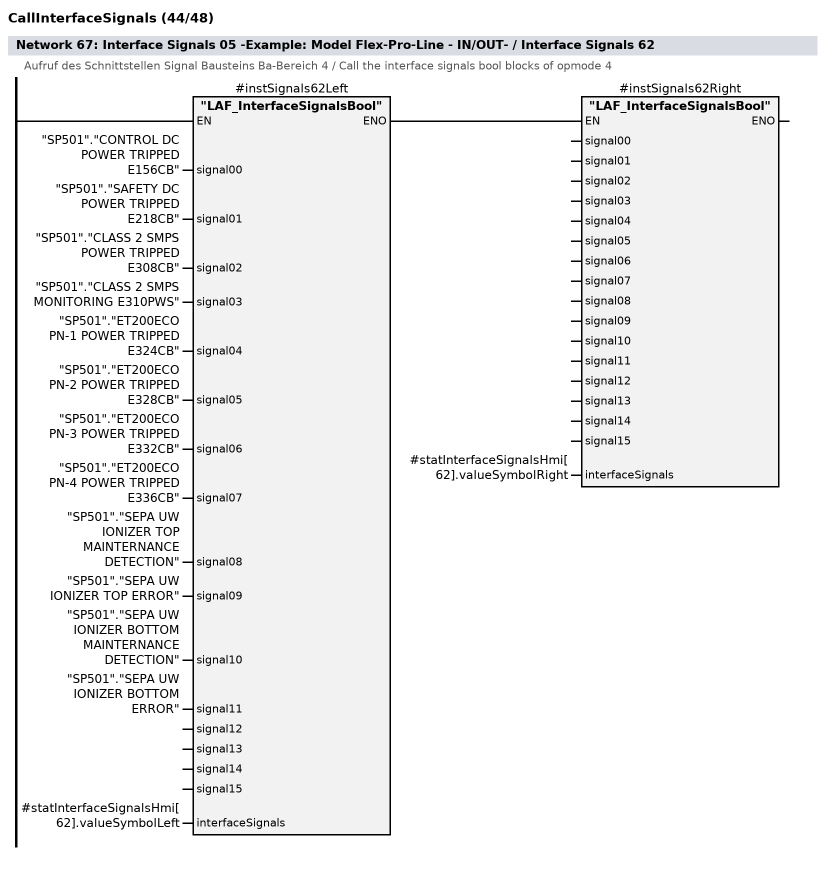
   RUNG wire#powerrail
      #instSignals62Left(signal00 := "SP501"."CONTROL DC POWER TRIPPED E156CB", signal01 := "SP501"."SAFETY DC POWER TRIPPED E218CB", signal02 := "SP501"."CLASS 2 SMPS POWER TRIPPED E308CB", signal03 := "SP501"."CLASS 2 SMPS MONITORING E310PWS", signal04 := "SP501"."ET200ECO PN-1 POWER TRIPPED E324CB", signal05 := "SP501"."ET200ECO PN-2 POWER TRIPPED E328CB", signal06 := "SP501"."ET200ECO PN-3 POWER TRIPPED E332CB", signal07 := "SP501"."ET200ECO PN-4 POWER TRIPPED E336CB", signal08 := "SP501"."SEPA UW IONIZER TOP MAINTERNANCE DETECTION", signal09 := "SP501"."SEPA UW IONIZER TOP ERROR", signal10 := "SP501"."SEPA UW IONIZER BOTTOM MAINTERNANCE DETECTION", signal11 := "SP501"."SEPA UW IONIZER BOTTOM ERROR", signal12 :=, signal13 :=, signal14 :=, signal15 :=, interfaceSignals := #statInterfaceSignalsHmi[62].valueSymbolLeft)
      #instSignals62Right(signal00 :=, signal01 :=, signal02 :=, signal03 :=, signal04 :=, signal05 :=, signal06 :=, signal07 :=, signal08 :=, signal09 :=, signal10 :=, signal11 :=, signal12 :=, signal13 :=, signal14 :=, signal15 :=, interfaceSignals := #statInterfaceSignalsHmi[62].valueSymbolRight)
   END_RUNG
   // the same network as SCL:
   #instSignals62Left(signal00 := "SP501"."CONTROL DC POWER TRIPPED E156CB",   // "LAF_InterfaceSignalsBool"
                      signal01 := "SP501"."SAFETY DC POWER TRIPPED E218CB",
                      signal02 := "SP501"."CLASS 2 SMPS POWER TRIPPED E308CB",
                      signal03 := "SP501"."CLASS 2 SMPS MONITORING E310PWS",
                      signal04 := "SP501"."ET200ECO PN-1 POWER TRIPPED E324CB",
                      signal05 := "SP501"."ET200ECO PN-2 POWER TRIPPED E328CB",
                      signal06 := "SP501"."ET200ECO PN-3 POWER TRIPPED E332CB",
                      signal07 := "SP501"."ET200ECO PN-4 POWER TRIPPED E336CB",
                      signal08 := "SP501"."SEPA UW IONIZER TOP MAINTERNANCE DETECTION",
                      signal09 := "SP501"."SEPA UW IONIZER TOP ERROR",
                      signal10 := "SP501"."SEPA UW IONIZER BOTTOM MAINTERNANCE DETECTION",
                      signal11 := "SP501"."SEPA UW IONIZER BOTTOM ERROR",
                      interfaceSignals := #statInterfaceSignalsHmi[62].valueSymbolLeft,
                      ENO => #_w1);
   IF #_w1 THEN
       #instSignals62Right(interfaceSignals := #statInterfaceSignalsHmi[62].valueSymbolRight);   // "LAF_InterfaceSignalsBool"
   END_IF;
END_REGION

REGION Network 68: Interface Signals 03 -Example: System flags & Clock flags- / Interface Signals63
   // Aufruf des Schnittstellen Signal Bausteins für die Systemvariablen / Call the interface signals bool blocks of system tags
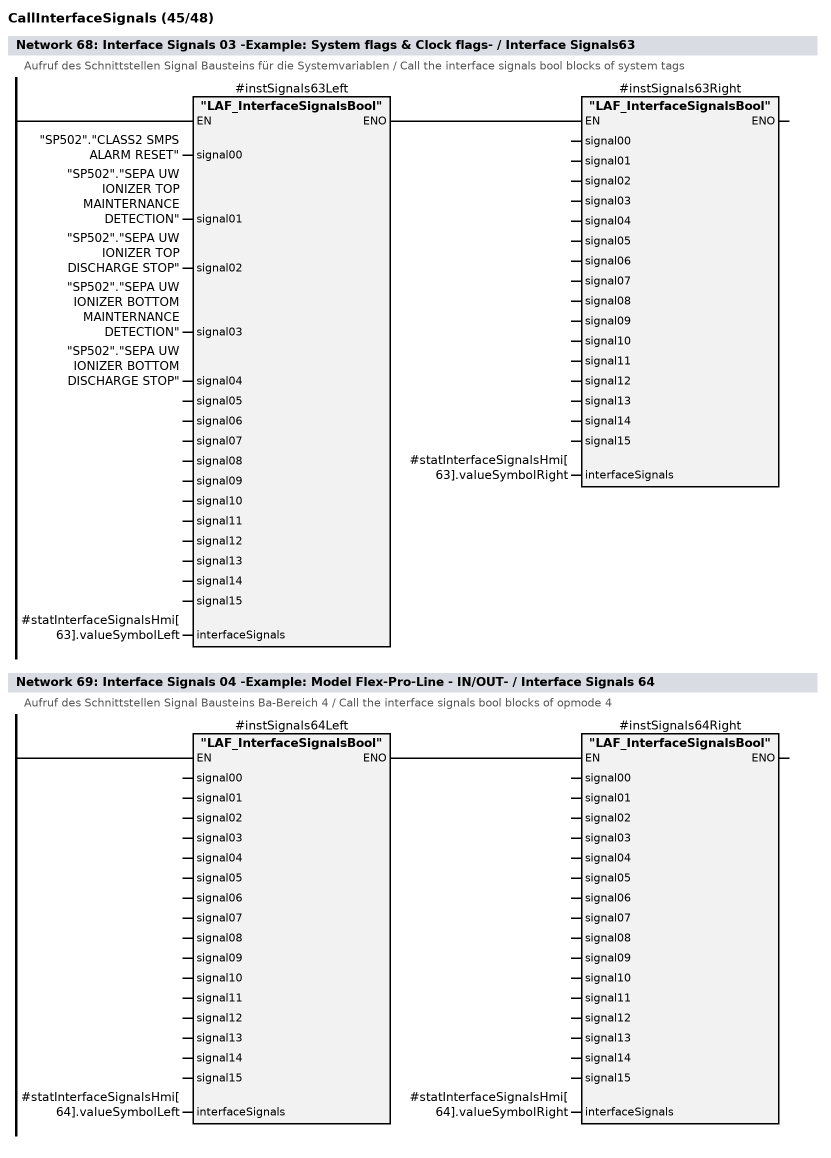
   RUNG wire#powerrail
      #instSignals63Left(signal00 := "SP502"."CLASS2 SMPS ALARM RESET", signal01 := "SP502"."SEPA UW IONIZER TOP MAINTERNANCE DETECTION", signal02 := "SP502"."SEPA UW IONIZER TOP DISCHARGE STOP", signal03 := "SP502"."SEPA UW IONIZER BOTTOM MAINTERNANCE DETECTION", signal04 := "SP502"."SEPA UW IONIZER BOTTOM DISCHARGE STOP", signal05 :=, signal06 :=, signal07 :=, signal08 :=, signal09 :=, signal10 :=, signal11 :=, signal12 :=, signal13 :=, signal14 :=, signal15 :=, interfaceSignals := #statInterfaceSignalsHmi[63].valueSymbolLeft)
      #instSignals63Right(signal00 :=, signal01 :=, signal02 :=, signal03 :=, signal04 :=, signal05 :=, signal06 :=, signal07 :=, signal08 :=, signal09 :=, signal10 :=, signal11 :=, signal12 :=, signal13 :=, signal14 :=, signal15 :=, interfaceSignals := #statInterfaceSignalsHmi[63].valueSymbolRight)
   END_RUNG
   // the same network as SCL:
   #instSignals63Left(signal00 := "SP502"."CLASS2 SMPS ALARM RESET",   // "LAF_InterfaceSignalsBool"
                      signal01 := "SP502"."SEPA UW IONIZER TOP MAINTERNANCE DETECTION",
                      signal02 := "SP502"."SEPA UW IONIZER TOP DISCHARGE STOP",
                      signal03 := "SP502"."SEPA UW IONIZER BOTTOM MAINTERNANCE DETECTION",
                      signal04 := "SP502"."SEPA UW IONIZER BOTTOM DISCHARGE STOP",
                      interfaceSignals := #statInterfaceSignalsHmi[63].valueSymbolLeft,
                      ENO => #_w1);
   IF #_w1 THEN
       #instSignals63Right(interfaceSignals := #statInterfaceSignalsHmi[63].valueSymbolRight);   // "LAF_InterfaceSignalsBool"
   END_IF;
END_REGION

REGION Network 69: Interface Signals 04 -Example: Model Flex-Pro-Line - IN/OUT- / Interface Signals 64
   // Aufruf des Schnittstellen Signal Bausteins Ba-Bereich 4 / Call the interface signals bool blocks of opmode 4
   RUNG wire#powerrail
      #instSignals64Left(signal00 :=, signal01 :=, signal02 :=, signal03 :=, signal04 :=, signal05 :=, signal06 :=, signal07 :=, signal08 :=, signal09 :=, signal10 :=, signal11 :=, signal12 :=, signal13 :=, signal14 :=, signal15 :=, interfaceSignals := #statInterfaceSignalsHmi[64].valueSymbolLeft)
      #instSignals64Right(signal00 :=, signal01 :=, signal02 :=, signal03 :=, signal04 :=, signal05 :=, signal06 :=, signal07 :=, signal08 :=, signal09 :=, signal10 :=, signal11 :=, signal12 :=, signal13 :=, signal14 :=, signal15 :=, interfaceSignals := #statInterfaceSignalsHmi[64].valueSymbolRight)
   END_RUNG
   // the same network as SCL:
   #instSignals64Left(interfaceSignals := #statInterfaceSignalsHmi[64].valueSymbolLeft, ENO => #_w1);   // "LAF_InterfaceSignalsBool"
   IF #_w1 THEN
       #instSignals64Right(interfaceSignals := #statInterfaceSignalsHmi[64].valueSymbolRight);   // "LAF_InterfaceSignalsBool"
   END_IF;
END_REGION

REGION Network 70: Interface Signals 05 -Example: Model Flex-Pro-Line - IN/OUT- / Interface Signals 65
   // Aufruf des Schnittstellen Signal Bausteins Ba-Bereich 4 / Call the interface signals bool blocks of opmode 4
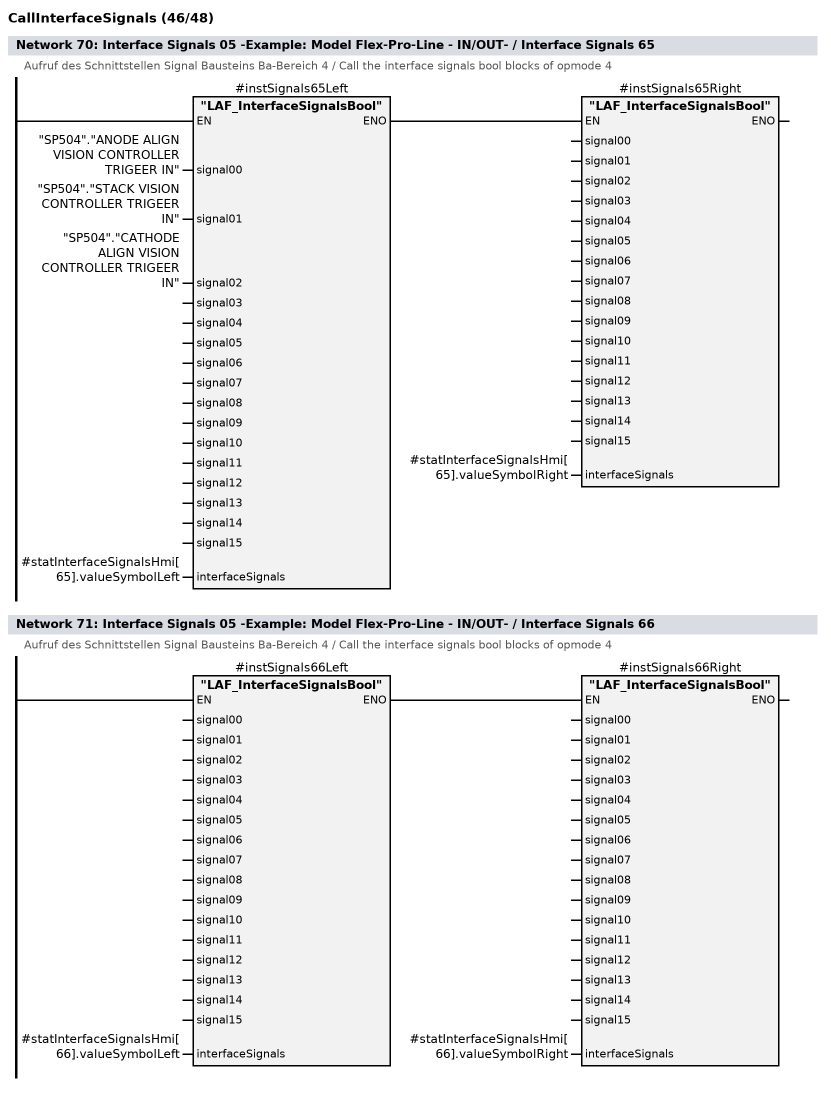
   RUNG wire#powerrail
      #instSignals65Left(signal00 := "SP504"."ANODE ALIGN VISION CONTROLLER TRIGEER IN", signal01 := "SP504"."STACK VISION CONTROLLER TRIGEER IN", signal02 := "SP504"."CATHODE ALIGN VISION CONTROLLER TRIGEER IN", signal03 :=, signal04 :=, signal05 :=, signal06 :=, signal07 :=, signal08 :=, signal09 :=, signal10 :=, signal11 :=, signal12 :=, signal13 :=, signal14 :=, signal15 :=, interfaceSignals := #statInterfaceSignalsHmi[65].valueSymbolLeft)
      #instSignals65Right(signal00 :=, signal01 :=, signal02 :=, signal03 :=, signal04 :=, signal05 :=, signal06 :=, signal07 :=, signal08 :=, signal09 :=, signal10 :=, signal11 :=, signal12 :=, signal13 :=, signal14 :=, signal15 :=, interfaceSignals := #statInterfaceSignalsHmi[65].valueSymbolRight)
   END_RUNG
   // the same network as SCL:
   #instSignals65Left(signal00 := "SP504"."ANODE ALIGN VISION CONTROLLER TRIGEER IN",   // "LAF_InterfaceSignalsBool"
                      signal01 := "SP504"."STACK VISION CONTROLLER TRIGEER IN",
                      signal02 := "SP504"."CATHODE ALIGN VISION CONTROLLER TRIGEER IN",
                      interfaceSignals := #statInterfaceSignalsHmi[65].valueSymbolLeft,
                      ENO => #_w1);
   IF #_w1 THEN
       #instSignals65Right(interfaceSignals := #statInterfaceSignalsHmi[65].valueSymbolRight);   // "LAF_InterfaceSignalsBool"
   END_IF;
END_REGION

REGION Network 71: Interface Signals 05 -Example: Model Flex-Pro-Line - IN/OUT- / Interface Signals 66
   // Aufruf des Schnittstellen Signal Bausteins Ba-Bereich 4 / Call the interface signals bool blocks of opmode 4
   RUNG wire#powerrail
      #instSignals66Left(signal00 :=, signal01 :=, signal02 :=, signal03 :=, signal04 :=, signal05 :=, signal06 :=, signal07 :=, signal08 :=, signal09 :=, signal10 :=, signal11 :=, signal12 :=, signal13 :=, signal14 :=, signal15 :=, interfaceSignals := #statInterfaceSignalsHmi[66].valueSymbolLeft)
      #instSignals66Right(signal00 :=, signal01 :=, signal02 :=, signal03 :=, signal04 :=, signal05 :=, signal06 :=, signal07 :=, signal08 :=, signal09 :=, signal10 :=, signal11 :=, signal12 :=, signal13 :=, signal14 :=, signal15 :=, interfaceSignals := #statInterfaceSignalsHmi[66].valueSymbolRight)
   END_RUNG
   // the same network as SCL:
   #instSignals66Left(interfaceSignals := #statInterfaceSignalsHmi[66].valueSymbolLeft, ENO => #_w1);   // "LAF_InterfaceSignalsBool"
   IF #_w1 THEN
       #instSignals66Right(interfaceSignals := #statInterfaceSignalsHmi[66].valueSymbolRight);   // "LAF_InterfaceSignalsBool"
   END_IF;
END_REGION

REGION Network 72: Interface Signals 05 -Example: Model Flex-Pro-Line - IN/OUT- / Interface Signals 67
   // Aufruf des Schnittstellen Signal Bausteins Ba-Bereich 4 / Call the interface signals bool blocks of opmode 4
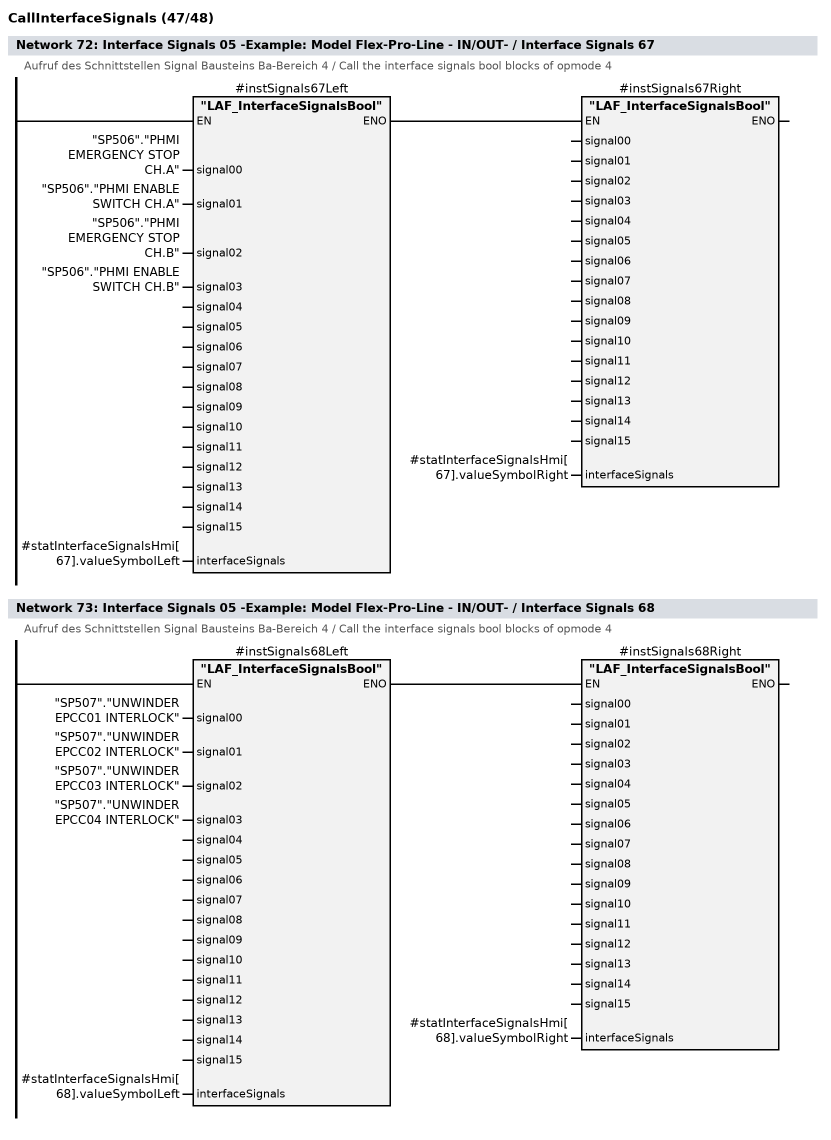
   RUNG wire#powerrail
      #instSignals67Left(signal00 := "SP506"."PHMI EMERGENCY STOP CH.A", signal01 := "SP506"."PHMI ENABLE SWITCH CH.A", signal02 := "SP506"."PHMI EMERGENCY STOP CH.B", signal03 := "SP506"."PHMI ENABLE SWITCH CH.B", signal04 :=, signal05 :=, signal06 :=, signal07 :=, signal08 :=, signal09 :=, signal10 :=, signal11 :=, signal12 :=, signal13 :=, signal14 :=, signal15 :=, interfaceSignals := #statInterfaceSignalsHmi[67].valueSymbolLeft)
      #instSignals67Right(signal00 :=, signal01 :=, signal02 :=, signal03 :=, signal04 :=, signal05 :=, signal06 :=, signal07 :=, signal08 :=, signal09 :=, signal10 :=, signal11 :=, signal12 :=, signal13 :=, signal14 :=, signal15 :=, interfaceSignals := #statInterfaceSignalsHmi[67].valueSymbolRight)
   END_RUNG
   // the same network as SCL:
   #instSignals67Left(signal00 := "SP506"."PHMI EMERGENCY STOP CH.A",   // "LAF_InterfaceSignalsBool"
                      signal01 := "SP506"."PHMI ENABLE SWITCH CH.A",
                      signal02 := "SP506"."PHMI EMERGENCY STOP CH.B",
                      signal03 := "SP506"."PHMI ENABLE SWITCH CH.B",
                      interfaceSignals := #statInterfaceSignalsHmi[67].valueSymbolLeft,
                      ENO => #_w1);
   IF #_w1 THEN
       #instSignals67Right(interfaceSignals := #statInterfaceSignalsHmi[67].valueSymbolRight);   // "LAF_InterfaceSignalsBool"
   END_IF;
END_REGION

REGION Network 73: Interface Signals 05 -Example: Model Flex-Pro-Line - IN/OUT- / Interface Signals 68
   // Aufruf des Schnittstellen Signal Bausteins Ba-Bereich 4 / Call the interface signals bool blocks of opmode 4
   RUNG wire#powerrail
      #instSignals68Left(signal00 := "SP507"."UNWINDER EPCC01 INTERLOCK", signal01 := "SP507"."UNWINDER EPCC02 INTERLOCK", signal02 := "SP507"."UNWINDER EPCC03 INTERLOCK", signal03 := "SP507"."UNWINDER EPCC04 INTERLOCK", signal04 :=, signal05 :=, signal06 :=, signal07 :=, signal08 :=, signal09 :=, signal10 :=, signal11 :=, signal12 :=, signal13 :=, signal14 :=, signal15 :=, interfaceSignals := #statInterfaceSignalsHmi[68].valueSymbolLeft)
      #instSignals68Right(signal00 :=, signal01 :=, signal02 :=, signal03 :=, signal04 :=, signal05 :=, signal06 :=, signal07 :=, signal08 :=, signal09 :=, signal10 :=, signal11 :=, signal12 :=, signal13 :=, signal14 :=, signal15 :=, interfaceSignals := #statInterfaceSignalsHmi[68].valueSymbolRight)
   END_RUNG
   // the same network as SCL:
   #instSignals68Left(signal00 := "SP507"."UNWINDER EPCC01 INTERLOCK",   // "LAF_InterfaceSignalsBool"
                      signal01 := "SP507"."UNWINDER EPCC02 INTERLOCK",
                      signal02 := "SP507"."UNWINDER EPCC03 INTERLOCK",
                      signal03 := "SP507"."UNWINDER EPCC04 INTERLOCK",
                      interfaceSignals := #statInterfaceSignalsHmi[68].valueSymbolLeft,
                      ENO => #_w1);
   IF #_w1 THEN
       #instSignals68Right(interfaceSignals := #statInterfaceSignalsHmi[68].valueSymbolRight);   // "LAF_InterfaceSignalsBool"
   END_IF;
END_REGION

REGION Network 74: Interface Signals 05 -Example: Model Flex-Pro-Line - IN/OUT- / Interface Signals 69
   // Aufruf des Schnittstellen Signal Bausteins Ba-Bereich 4 / Call the interface signals bool blocks of opmode 4
